REGION Network 92: Step[1902] :
   RUNG wire#powerrail
      { S7_Templates := "SrcType := DInt" } EQ_Contact(in1 := "Unit1.Em2.ControlNodes".semiAutoSplice.sequence.status.currentStep, in2 := #JOB_19_STEP_02)
      Contact( "Unit1.Em2.ControlNodes".semiAutoSplice.sequence.status.seqActive )
      wire#w1
      Coil( "Unit1.Em2.ControlNodes".semiAutoSplice."step".action1[1902] )
   END_RUNG
   RUNG wire#w1
      Coil( "Unit1.Em2.ControlNodes".semiAutoSplice."step".transition1[1902] )
   END_RUNG
   RUNG wire#w1
      Contact( "Unit1.Em2.ControlNodes".semiAutoSplice."step".transition1[1902] )
      { S7_Templates := "time_type := Time" } #statTonTimer[1902].TON(pt := #SeqDelayTime, et =>)
      Move(in := #JOB_19_STEP_03, out1 => "Unit1.Em2.ControlNodes".semiAutoSplice.sequence.status.nextStep)
   END_RUNG
   // the same network as SCL:
   "Unit1.Em2.ControlNodes".semiAutoSplice."step".action1[1902] := ("Unit1.Em2.ControlNodes".semiAutoSplice.sequence.status.currentStep = #JOB_19_STEP_02) AND "Unit1.Em2.ControlNodes".semiAutoSplice.sequence.status.seqActive;
   "Unit1.Em2.ControlNodes".semiAutoSplice."step".transition1[1902] := ("Unit1.Em2.ControlNodes".semiAutoSplice.sequence.status.currentStep = #JOB_19_STEP_02) AND "Unit1.Em2.ControlNodes".semiAutoSplice.sequence.status.seqActive;
   #statTonTimer[1902].TON(IN := ("Unit1.Em2.ControlNodes".semiAutoSplice.sequence.status.currentStep = #JOB_19_STEP_02) AND "Unit1.Em2.ControlNodes".semiAutoSplice.sequence.status.seqActive AND "Unit1.Em2.ControlNodes".semiAutoSplice."step".transition1[1902],
                           PT := #SeqDelayTime);
   IF #statTonTimer[1902].Q THEN
       "Unit1.Em2.ControlNodes".semiAutoSplice.sequence.status.nextStep := #JOB_19_STEP_03;
   END_IF;
END_REGION

REGION Network 93: Step[1903] :
   RUNG wire#powerrail
      { S7_Templates := "SrcType := DInt" } EQ_Contact(in1 := "Unit1.Em2.ControlNodes".semiAutoSplice.sequence.status.currentStep, in2 := #JOB_19_STEP_03)
      Contact( "Unit1.Em2.ControlNodes".semiAutoSplice.sequence.status.seqActive )
      wire#w1
      Coil( "Unit1.Em2.ControlNodes".semiAutoSplice."step".action1[1903] )
   END_RUNG
   RUNG wire#w1
      Coil( "Unit1.Em2.ControlNodes".semiAutoSplice."step".transition1[1903] )
   END_RUNG
   RUNG wire#w1
      Contact( "Unit1.Em2.ControlNodes".semiAutoSplice."step".transition1[1903] )
      { S7_Templates := "time_type := Time" } #statTonTimer[1903].TON(pt := #SeqDelayTime, et =>)
      Move(in := #JOB_19_STEP_04, out1 => "Unit1.Em2.ControlNodes".semiAutoSplice.sequence.status.nextStep)
   END_RUNG
   // the same network as SCL:
   "Unit1.Em2.ControlNodes".semiAutoSplice."step".action1[1903] := ("Unit1.Em2.ControlNodes".semiAutoSplice.sequence.status.currentStep = #JOB_19_STEP_03) AND "Unit1.Em2.ControlNodes".semiAutoSplice.sequence.status.seqActive;
   "Unit1.Em2.ControlNodes".semiAutoSplice."step".transition1[1903] := ("Unit1.Em2.ControlNodes".semiAutoSplice.sequence.status.currentStep = #JOB_19_STEP_03) AND "Unit1.Em2.ControlNodes".semiAutoSplice.sequence.status.seqActive;
   #statTonTimer[1903].TON(IN := ("Unit1.Em2.ControlNodes".semiAutoSplice.sequence.status.currentStep = #JOB_19_STEP_03) AND "Unit1.Em2.ControlNodes".semiAutoSplice.sequence.status.seqActive AND "Unit1.Em2.ControlNodes".semiAutoSplice."step".transition1[1903],
                           PT := #SeqDelayTime);
   IF #statTonTimer[1903].Q THEN
       "Unit1.Em2.ControlNodes".semiAutoSplice.sequence.status.nextStep := #JOB_19_STEP_04;
   END_IF;
END_REGION

REGION Network 94: Step[1904] :
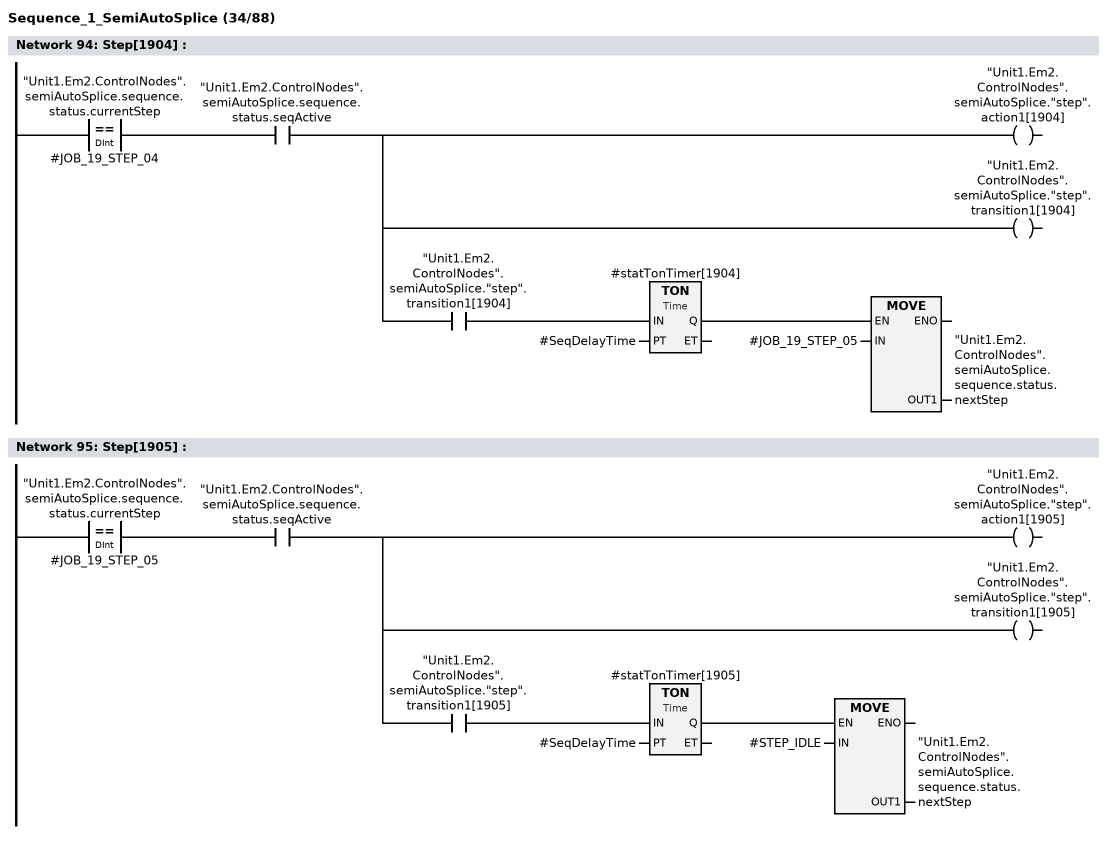
   RUNG wire#powerrail
      { S7_Templates := "SrcType := DInt" } EQ_Contact(in1 := "Unit1.Em2.ControlNodes".semiAutoSplice.sequence.status.currentStep, in2 := #JOB_19_STEP_04)
      Contact( "Unit1.Em2.ControlNodes".semiAutoSplice.sequence.status.seqActive )
      wire#w1
      Coil( "Unit1.Em2.ControlNodes".semiAutoSplice."step".action1[1904] )
   END_RUNG
   RUNG wire#w1
      Coil( "Unit1.Em2.ControlNodes".semiAutoSplice."step".transition1[1904] )
   END_RUNG
   RUNG wire#w1
      Contact( "Unit1.Em2.ControlNodes".semiAutoSplice."step".transition1[1904] )
      { S7_Templates := "time_type := Time" } #statTonTimer[1904].TON(pt := #SeqDelayTime, et =>)
      Move(in := #JOB_19_STEP_05, out1 => "Unit1.Em2.ControlNodes".semiAutoSplice.sequence.status.nextStep)
   END_RUNG
   // the same network as SCL:
   "Unit1.Em2.ControlNodes".semiAutoSplice."step".action1[1904] := ("Unit1.Em2.ControlNodes".semiAutoSplice.sequence.status.currentStep = #JOB_19_STEP_04) AND "Unit1.Em2.ControlNodes".semiAutoSplice.sequence.status.seqActive;
   "Unit1.Em2.ControlNodes".semiAutoSplice."step".transition1[1904] := ("Unit1.Em2.ControlNodes".semiAutoSplice.sequence.status.currentStep = #JOB_19_STEP_04) AND "Unit1.Em2.ControlNodes".semiAutoSplice.sequence.status.seqActive;
   #statTonTimer[1904].TON(IN := ("Unit1.Em2.ControlNodes".semiAutoSplice.sequence.status.currentStep = #JOB_19_STEP_04) AND "Unit1.Em2.ControlNodes".semiAutoSplice.sequence.status.seqActive AND "Unit1.Em2.ControlNodes".semiAutoSplice."step".transition1[1904],
                           PT := #SeqDelayTime);
   IF #statTonTimer[1904].Q THEN
       "Unit1.Em2.ControlNodes".semiAutoSplice.sequence.status.nextStep := #JOB_19_STEP_05;
   END_IF;
END_REGION

REGION Network 95: Step[1905] :
   RUNG wire#powerrail
      { S7_Templates := "SrcType := DInt" } EQ_Contact(in1 := "Unit1.Em2.ControlNodes".semiAutoSplice.sequence.status.currentStep, in2 := #JOB_19_STEP_05)
      Contact( "Unit1.Em2.ControlNodes".semiAutoSplice.sequence.status.seqActive )
      wire#w1
      Coil( "Unit1.Em2.ControlNodes".semiAutoSplice."step".action1[1905] )
   END_RUNG
   RUNG wire#w1
      Coil( "Unit1.Em2.ControlNodes".semiAutoSplice."step".transition1[1905] )
   END_RUNG
   RUNG wire#w1
      Contact( "Unit1.Em2.ControlNodes".semiAutoSplice."step".transition1[1905] )
      { S7_Templates := "time_type := Time" } #statTonTimer[1905].TON(pt := #SeqDelayTime, et =>)
      Move(in := #STEP_IDLE, out1 => "Unit1.Em2.ControlNodes".semiAutoSplice.sequence.status.nextStep)
   END_RUNG
   // the same network as SCL:
   "Unit1.Em2.ControlNodes".semiAutoSplice."step".action1[1905] := ("Unit1.Em2.ControlNodes".semiAutoSplice.sequence.status.currentStep = #JOB_19_STEP_05) AND "Unit1.Em2.ControlNodes".semiAutoSplice.sequence.status.seqActive;
   "Unit1.Em2.ControlNodes".semiAutoSplice."step".transition1[1905] := ("Unit1.Em2.ControlNodes".semiAutoSplice.sequence.status.currentStep = #JOB_19_STEP_05) AND "Unit1.Em2.ControlNodes".semiAutoSplice.sequence.status.seqActive;
   #statTonTimer[1905].TON(IN := ("Unit1.Em2.ControlNodes".semiAutoSplice.sequence.status.currentStep = #JOB_19_STEP_05) AND "Unit1.Em2.ControlNodes".semiAutoSplice.sequence.status.seqActive AND "Unit1.Em2.ControlNodes".semiAutoSplice."step".transition1[1905],
                           PT := #SeqDelayTime);
   IF #statTonTimer[1905].Q THEN
       "Unit1.Em2.ControlNodes".semiAutoSplice.sequence.status.nextStep := #STEP_IDLE;
   END_IF;
END_REGION

REGION Network 96: Step[2001] : Pad Btm Link Btm Left/right Vacc Off (Top Left/Right Vacc On)
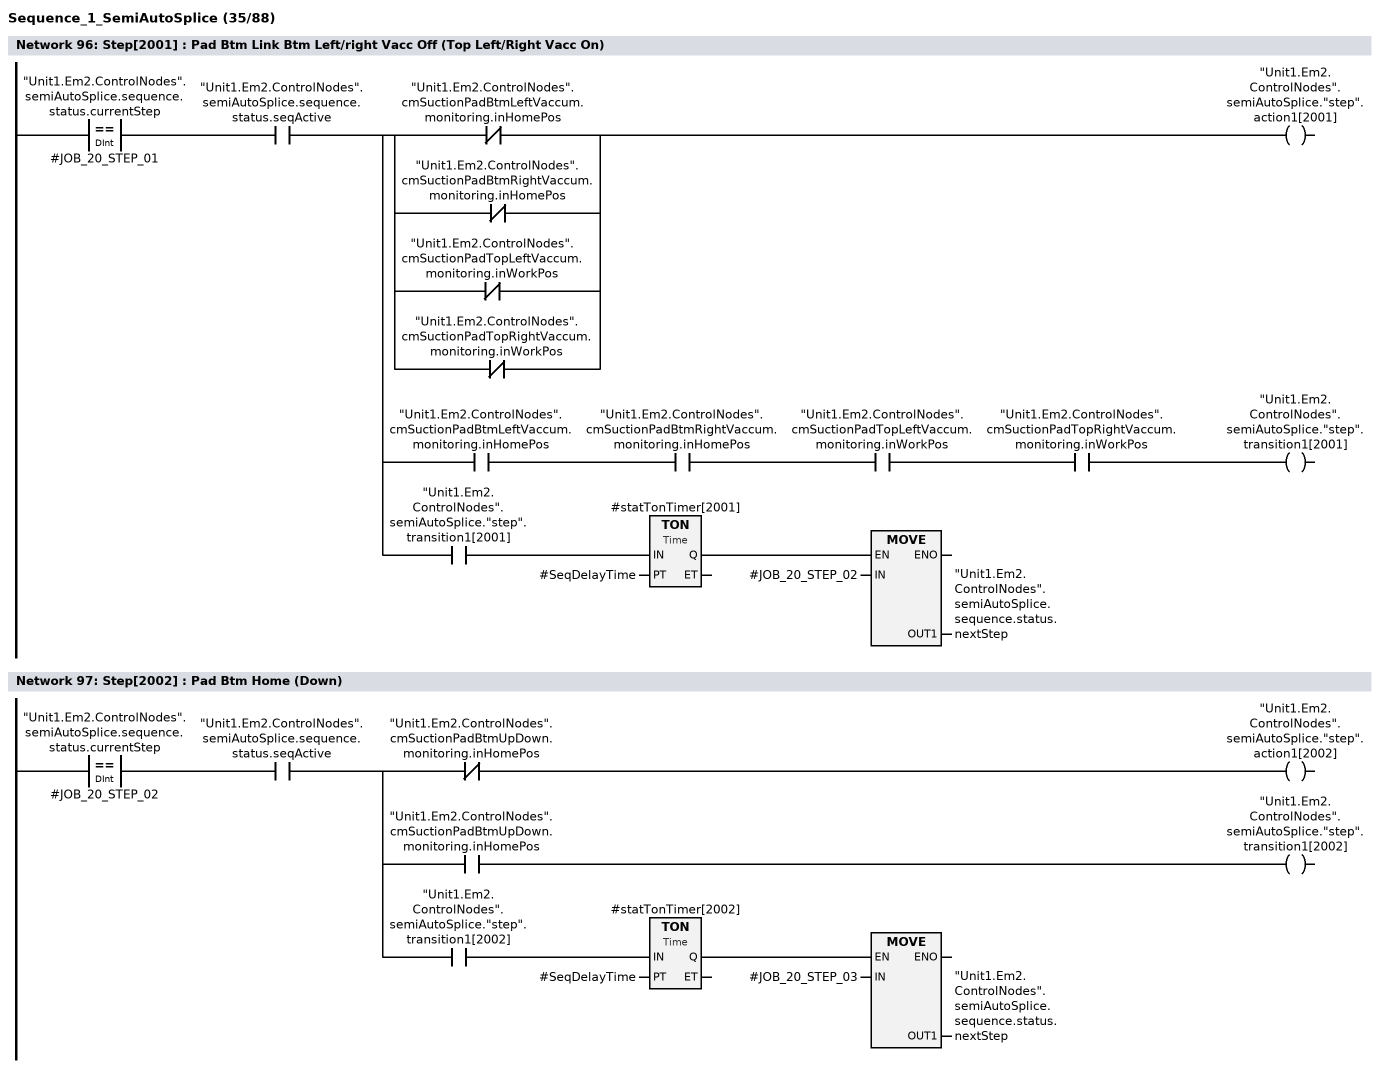
   RUNG wire#powerrail
      { S7_Templates := "SrcType := DInt" } EQ_Contact(in1 := "Unit1.Em2.ControlNodes".semiAutoSplice.sequence.status.currentStep, in2 := #JOB_20_STEP_01)
      Contact( "Unit1.Em2.ControlNodes".semiAutoSplice.sequence.status.seqActive )
      wire#w1
      I_Contact( "Unit1.Em2.ControlNodes".cmSuctionPadBtmLeftVaccum.monitoring.inHomePos )
      wire#w2
      Coil( "Unit1.Em2.ControlNodes".semiAutoSplice."step".action1[2001] )
   END_RUNG
   RUNG wire#w1
      I_Contact( "Unit1.Em2.ControlNodes".cmSuctionPadBtmRightVaccum.monitoring.inHomePos )
   END_RUNG wire#w2
   RUNG wire#w1
      I_Contact( "Unit1.Em2.ControlNodes".cmSuctionPadTopLeftVaccum.monitoring.inWorkPos )
   END_RUNG wire#w2
   RUNG wire#w1
      I_Contact( "Unit1.Em2.ControlNodes".cmSuctionPadTopRightVaccum.monitoring.inWorkPos )
   END_RUNG wire#w2
   RUNG wire#w1
      Contact( "Unit1.Em2.ControlNodes".cmSuctionPadBtmLeftVaccum.monitoring.inHomePos )
      Contact( "Unit1.Em2.ControlNodes".cmSuctionPadBtmRightVaccum.monitoring.inHomePos )
      Contact( "Unit1.Em2.ControlNodes".cmSuctionPadTopLeftVaccum.monitoring.inWorkPos )
      Contact( "Unit1.Em2.ControlNodes".cmSuctionPadTopRightVaccum.monitoring.inWorkPos )
      Coil( "Unit1.Em2.ControlNodes".semiAutoSplice."step".transition1[2001] )
   END_RUNG
   RUNG wire#w1
      Contact( "Unit1.Em2.ControlNodes".semiAutoSplice."step".transition1[2001] )
      { S7_Templates := "time_type := Time" } #statTonTimer[2001].TON(pt := #SeqDelayTime, et =>)
      Move(in := #JOB_20_STEP_02, out1 => "Unit1.Em2.ControlNodes".semiAutoSplice.sequence.status.nextStep)
   END_RUNG
   // the same network as SCL:
   #_w1 := ("Unit1.Em2.ControlNodes".semiAutoSplice.sequence.status.currentStep = #JOB_20_STEP_01) AND "Unit1.Em2.ControlNodes".semiAutoSplice.sequence.status.seqActive;
   "Unit1.Em2.ControlNodes".semiAutoSplice."step".action1[2001] := #_w1 AND (NOT "Unit1.Em2.ControlNodes".cmSuctionPadBtmLeftVaccum.monitoring.inHomePos OR NOT "Unit1.Em2.ControlNodes".cmSuctionPadBtmRightVaccum.monitoring.inHomePos OR NOT "Unit1.Em2.ControlNodes".cmSuctionPadTopLeftVaccum.monitoring.inWorkPos OR NOT "Unit1.Em2.ControlNodes".cmSuctionPadTopRightVaccum.monitoring.inWorkPos);
   "Unit1.Em2.ControlNodes".semiAutoSplice."step".transition1[2001] := #_w1 AND "Unit1.Em2.ControlNodes".cmSuctionPadBtmLeftVaccum.monitoring.inHomePos AND "Unit1.Em2.ControlNodes".cmSuctionPadBtmRightVaccum.monitoring.inHomePos AND "Unit1.Em2.ControlNodes".cmSuctionPadTopLeftVaccum.monitoring.inWorkPos AND "Unit1.Em2.ControlNodes".cmSuctionPadTopRightVaccum.monitoring.inWorkPos;
   #statTonTimer[2001].TON(IN := #_w1 AND "Unit1.Em2.ControlNodes".semiAutoSplice."step".transition1[2001],
                           PT := #SeqDelayTime);
   IF #statTonTimer[2001].Q THEN
       "Unit1.Em2.ControlNodes".semiAutoSplice.sequence.status.nextStep := #JOB_20_STEP_02;
   END_IF;
END_REGION

REGION Network 97: Step[2002] : Pad Btm Home (Down)
   RUNG wire#powerrail
      { S7_Templates := "SrcType := DInt" } EQ_Contact(in1 := "Unit1.Em2.ControlNodes".semiAutoSplice.sequence.status.currentStep, in2 := #JOB_20_STEP_02)
      Contact( "Unit1.Em2.ControlNodes".semiAutoSplice.sequence.status.seqActive )
      wire#w1
      I_Contact( "Unit1.Em2.ControlNodes".cmSuctionPadBtmUpDown.monitoring.inHomePos )
      Coil( "Unit1.Em2.ControlNodes".semiAutoSplice."step".action1[2002] )
   END_RUNG
   RUNG wire#w1
      Contact( "Unit1.Em2.ControlNodes".cmSuctionPadBtmUpDown.monitoring.inHomePos )
      Coil( "Unit1.Em2.ControlNodes".semiAutoSplice."step".transition1[2002] )
   END_RUNG
   RUNG wire#w1
      Contact( "Unit1.Em2.ControlNodes".semiAutoSplice."step".transition1[2002] )
      { S7_Templates := "time_type := Time" } #statTonTimer[2002].TON(pt := #SeqDelayTime, et =>)
      Move(in := #JOB_20_STEP_03, out1 => "Unit1.Em2.ControlNodes".semiAutoSplice.sequence.status.nextStep)
   END_RUNG
   // the same network as SCL:
   #_w1 := ("Unit1.Em2.ControlNodes".semiAutoSplice.sequence.status.currentStep = #JOB_20_STEP_02) AND "Unit1.Em2.ControlNodes".semiAutoSplice.sequence.status.seqActive;
   "Unit1.Em2.ControlNodes".semiAutoSplice."step".action1[2002] := #_w1 AND NOT "Unit1.Em2.ControlNodes".cmSuctionPadBtmUpDown.monitoring.inHomePos;
   "Unit1.Em2.ControlNodes".semiAutoSplice."step".transition1[2002] := #_w1 AND "Unit1.Em2.ControlNodes".cmSuctionPadBtmUpDown.monitoring.inHomePos;
   #statTonTimer[2002].TON(IN := #_w1 AND "Unit1.Em2.ControlNodes".semiAutoSplice."step".transition1[2002],
                           PT := #SeqDelayTime);
   IF #statTonTimer[2002].Q THEN
       "Unit1.Em2.ControlNodes".semiAutoSplice.sequence.status.nextStep := #JOB_20_STEP_03;
   END_IF;
END_REGION

REGION Network 98: Step[2003] :
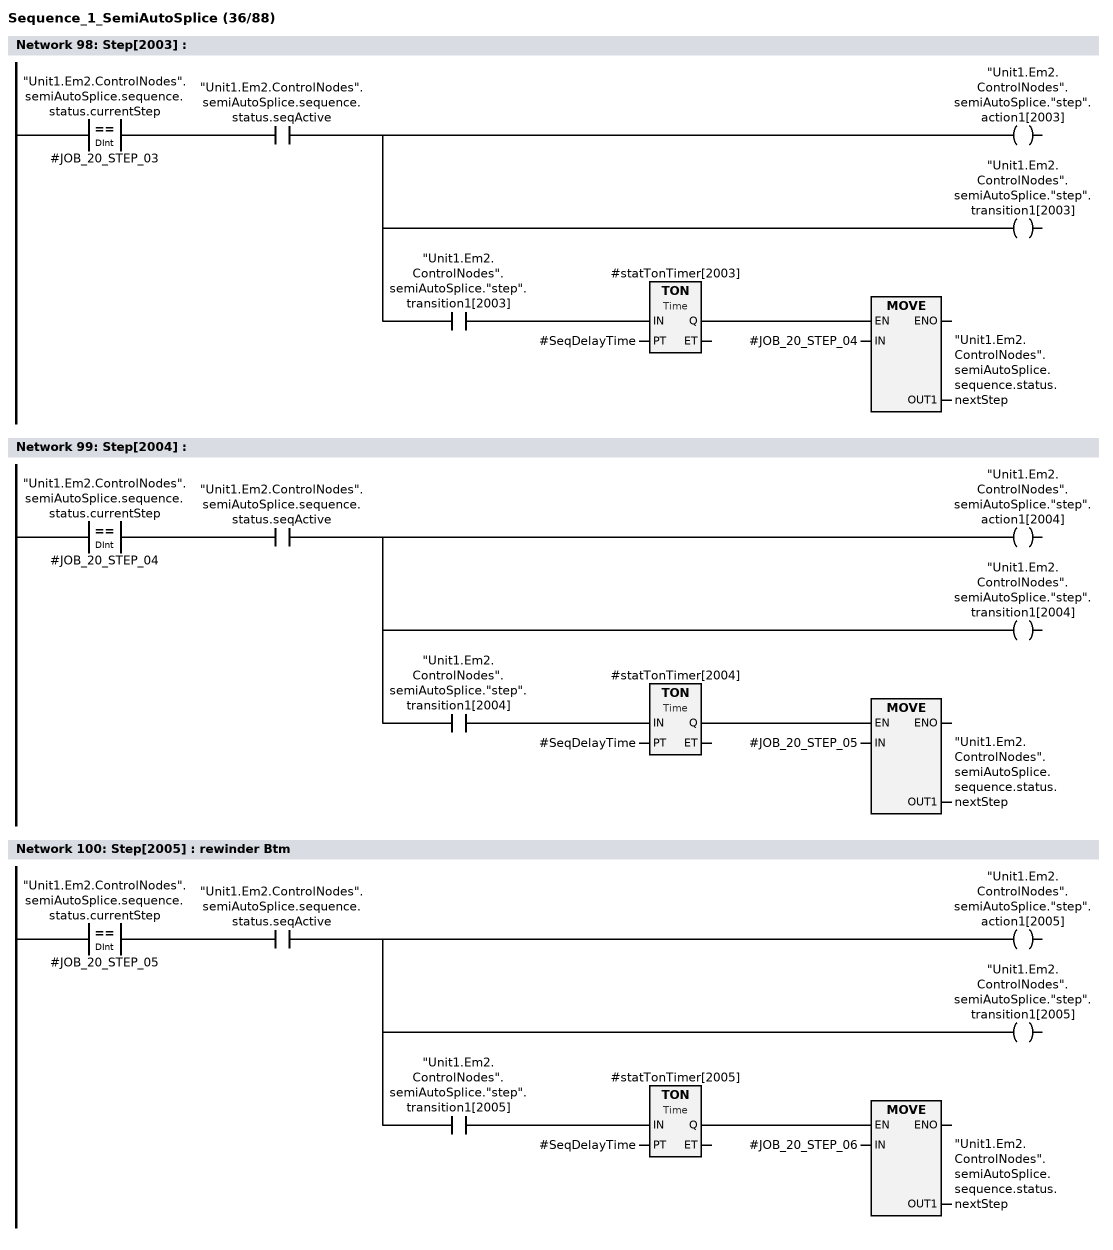
   RUNG wire#powerrail
      { S7_Templates := "SrcType := DInt" } EQ_Contact(in1 := "Unit1.Em2.ControlNodes".semiAutoSplice.sequence.status.currentStep, in2 := #JOB_20_STEP_03)
      Contact( "Unit1.Em2.ControlNodes".semiAutoSplice.sequence.status.seqActive )
      wire#w1
      Coil( "Unit1.Em2.ControlNodes".semiAutoSplice."step".action1[2003] )
   END_RUNG
   RUNG wire#w1
      Coil( "Unit1.Em2.ControlNodes".semiAutoSplice."step".transition1[2003] )
   END_RUNG
   RUNG wire#w1
      Contact( "Unit1.Em2.ControlNodes".semiAutoSplice."step".transition1[2003] )
      { S7_Templates := "time_type := Time" } #statTonTimer[2003].TON(pt := #SeqDelayTime, et =>)
      Move(in := #JOB_20_STEP_04, out1 => "Unit1.Em2.ControlNodes".semiAutoSplice.sequence.status.nextStep)
   END_RUNG
   // the same network as SCL:
   "Unit1.Em2.ControlNodes".semiAutoSplice."step".action1[2003] := ("Unit1.Em2.ControlNodes".semiAutoSplice.sequence.status.currentStep = #JOB_20_STEP_03) AND "Unit1.Em2.ControlNodes".semiAutoSplice.sequence.status.seqActive;
   "Unit1.Em2.ControlNodes".semiAutoSplice."step".transition1[2003] := ("Unit1.Em2.ControlNodes".semiAutoSplice.sequence.status.currentStep = #JOB_20_STEP_03) AND "Unit1.Em2.ControlNodes".semiAutoSplice.sequence.status.seqActive;
   #statTonTimer[2003].TON(IN := ("Unit1.Em2.ControlNodes".semiAutoSplice.sequence.status.currentStep = #JOB_20_STEP_03) AND "Unit1.Em2.ControlNodes".semiAutoSplice.sequence.status.seqActive AND "Unit1.Em2.ControlNodes".semiAutoSplice."step".transition1[2003],
                           PT := #SeqDelayTime);
   IF #statTonTimer[2003].Q THEN
       "Unit1.Em2.ControlNodes".semiAutoSplice.sequence.status.nextStep := #JOB_20_STEP_04;
   END_IF;
END_REGION

REGION Network 99: Step[2004] :
   RUNG wire#powerrail
      { S7_Templates := "SrcType := DInt" } EQ_Contact(in1 := "Unit1.Em2.ControlNodes".semiAutoSplice.sequence.status.currentStep, in2 := #JOB_20_STEP_04)
      Contact( "Unit1.Em2.ControlNodes".semiAutoSplice.sequence.status.seqActive )
      wire#w1
      Coil( "Unit1.Em2.ControlNodes".semiAutoSplice."step".action1[2004] )
   END_RUNG
   RUNG wire#w1
      Coil( "Unit1.Em2.ControlNodes".semiAutoSplice."step".transition1[2004] )
   END_RUNG
   RUNG wire#w1
      Contact( "Unit1.Em2.ControlNodes".semiAutoSplice."step".transition1[2004] )
      { S7_Templates := "time_type := Time" } #statTonTimer[2004].TON(pt := #SeqDelayTime, et =>)
      Move(in := #JOB_20_STEP_05, out1 => "Unit1.Em2.ControlNodes".semiAutoSplice.sequence.status.nextStep)
   END_RUNG
   // the same network as SCL:
   "Unit1.Em2.ControlNodes".semiAutoSplice."step".action1[2004] := ("Unit1.Em2.ControlNodes".semiAutoSplice.sequence.status.currentStep = #JOB_20_STEP_04) AND "Unit1.Em2.ControlNodes".semiAutoSplice.sequence.status.seqActive;
   "Unit1.Em2.ControlNodes".semiAutoSplice."step".transition1[2004] := ("Unit1.Em2.ControlNodes".semiAutoSplice.sequence.status.currentStep = #JOB_20_STEP_04) AND "Unit1.Em2.ControlNodes".semiAutoSplice.sequence.status.seqActive;
   #statTonTimer[2004].TON(IN := ("Unit1.Em2.ControlNodes".semiAutoSplice.sequence.status.currentStep = #JOB_20_STEP_04) AND "Unit1.Em2.ControlNodes".semiAutoSplice.sequence.status.seqActive AND "Unit1.Em2.ControlNodes".semiAutoSplice."step".transition1[2004],
                           PT := #SeqDelayTime);
   IF #statTonTimer[2004].Q THEN
       "Unit1.Em2.ControlNodes".semiAutoSplice.sequence.status.nextStep := #JOB_20_STEP_05;
   END_IF;
END_REGION

REGION Network 100: Step[2005] : rewinder Btm
   RUNG wire#powerrail
      { S7_Templates := "SrcType := DInt" } EQ_Contact(in1 := "Unit1.Em2.ControlNodes".semiAutoSplice.sequence.status.currentStep, in2 := #JOB_20_STEP_05)
      Contact( "Unit1.Em2.ControlNodes".semiAutoSplice.sequence.status.seqActive )
      wire#w1
      Coil( "Unit1.Em2.ControlNodes".semiAutoSplice."step".action1[2005] )
   END_RUNG
   RUNG wire#w1
      Coil( "Unit1.Em2.ControlNodes".semiAutoSplice."step".transition1[2005] )
   END_RUNG
   RUNG wire#w1
      Contact( "Unit1.Em2.ControlNodes".semiAutoSplice."step".transition1[2005] )
      { S7_Templates := "time_type := Time" } #statTonTimer[2005].TON(pt := #SeqDelayTime, et =>)
      Move(in := #JOB_20_STEP_06, out1 => "Unit1.Em2.ControlNodes".semiAutoSplice.sequence.status.nextStep)
   END_RUNG
   // the same network as SCL:
   "Unit1.Em2.ControlNodes".semiAutoSplice."step".action1[2005] := ("Unit1.Em2.ControlNodes".semiAutoSplice.sequence.status.currentStep = #JOB_20_STEP_05) AND "Unit1.Em2.ControlNodes".semiAutoSplice.sequence.status.seqActive;
   "Unit1.Em2.ControlNodes".semiAutoSplice."step".transition1[2005] := ("Unit1.Em2.ControlNodes".semiAutoSplice.sequence.status.currentStep = #JOB_20_STEP_05) AND "Unit1.Em2.ControlNodes".semiAutoSplice.sequence.status.seqActive;
   #statTonTimer[2005].TON(IN := ("Unit1.Em2.ControlNodes".semiAutoSplice.sequence.status.currentStep = #JOB_20_STEP_05) AND "Unit1.Em2.ControlNodes".semiAutoSplice.sequence.status.seqActive AND "Unit1.Em2.ControlNodes".semiAutoSplice."step".transition1[2005],
                           PT := #SeqDelayTime);
   IF #statTonTimer[2005].Q THEN
       "Unit1.Em2.ControlNodes".semiAutoSplice.sequence.status.nextStep := #JOB_20_STEP_06;
   END_IF;
END_REGION

REGION Network 101: Step[2006] : Complete
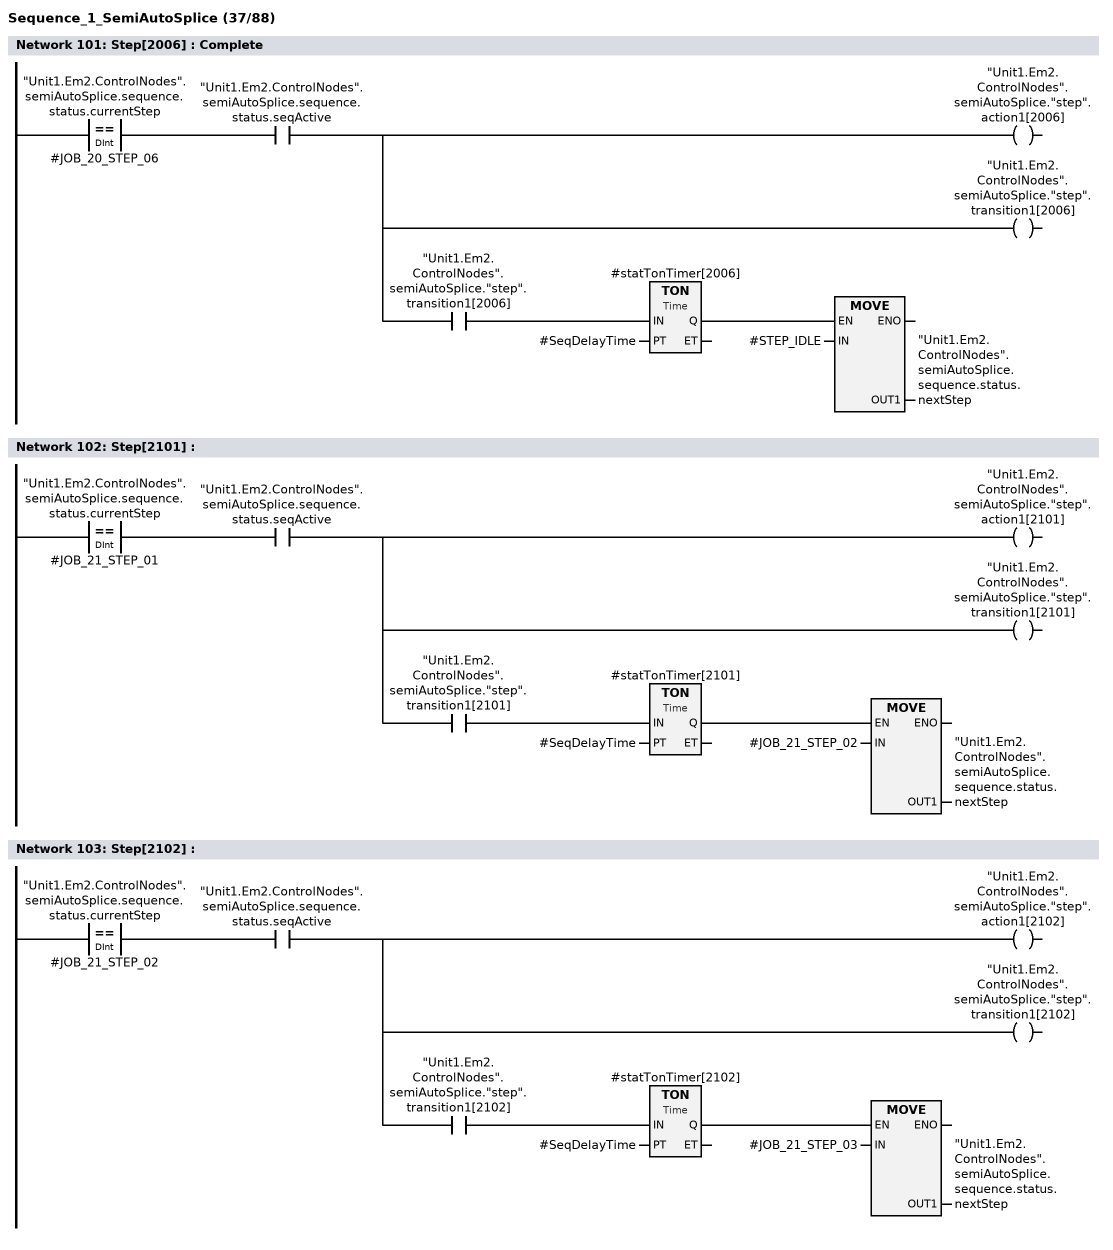
   RUNG wire#powerrail
      { S7_Templates := "SrcType := DInt" } EQ_Contact(in1 := "Unit1.Em2.ControlNodes".semiAutoSplice.sequence.status.currentStep, in2 := #JOB_20_STEP_06)
      Contact( "Unit1.Em2.ControlNodes".semiAutoSplice.sequence.status.seqActive )
      wire#w1
      Coil( "Unit1.Em2.ControlNodes".semiAutoSplice."step".action1[2006] )
   END_RUNG
   RUNG wire#w1
      Coil( "Unit1.Em2.ControlNodes".semiAutoSplice."step".transition1[2006] )
   END_RUNG
   RUNG wire#w1
      Contact( "Unit1.Em2.ControlNodes".semiAutoSplice."step".transition1[2006] )
      { S7_Templates := "time_type := Time" } #statTonTimer[2006].TON(pt := #SeqDelayTime, et =>)
      Move(in := #STEP_IDLE, out1 => "Unit1.Em2.ControlNodes".semiAutoSplice.sequence.status.nextStep)
   END_RUNG
   // the same network as SCL:
   "Unit1.Em2.ControlNodes".semiAutoSplice."step".action1[2006] := ("Unit1.Em2.ControlNodes".semiAutoSplice.sequence.status.currentStep = #JOB_20_STEP_06) AND "Unit1.Em2.ControlNodes".semiAutoSplice.sequence.status.seqActive;
   "Unit1.Em2.ControlNodes".semiAutoSplice."step".transition1[2006] := ("Unit1.Em2.ControlNodes".semiAutoSplice.sequence.status.currentStep = #JOB_20_STEP_06) AND "Unit1.Em2.ControlNodes".semiAutoSplice.sequence.status.seqActive;
   #statTonTimer[2006].TON(IN := ("Unit1.Em2.ControlNodes".semiAutoSplice.sequence.status.currentStep = #JOB_20_STEP_06) AND "Unit1.Em2.ControlNodes".semiAutoSplice.sequence.status.seqActive AND "Unit1.Em2.ControlNodes".semiAutoSplice."step".transition1[2006],
                           PT := #SeqDelayTime);
   IF #statTonTimer[2006].Q THEN
       "Unit1.Em2.ControlNodes".semiAutoSplice.sequence.status.nextStep := #STEP_IDLE;
   END_IF;
END_REGION

REGION Network 102: Step[2101] :
   RUNG wire#powerrail
      { S7_Templates := "SrcType := DInt" } EQ_Contact(in1 := "Unit1.Em2.ControlNodes".semiAutoSplice.sequence.status.currentStep, in2 := #JOB_21_STEP_01)
      Contact( "Unit1.Em2.ControlNodes".semiAutoSplice.sequence.status.seqActive )
      wire#w1
      Coil( "Unit1.Em2.ControlNodes".semiAutoSplice."step".action1[2101] )
   END_RUNG
   RUNG wire#w1
      Coil( "Unit1.Em2.ControlNodes".semiAutoSplice."step".transition1[2101] )
   END_RUNG
   RUNG wire#w1
      Contact( "Unit1.Em2.ControlNodes".semiAutoSplice."step".transition1[2101] )
      { S7_Templates := "time_type := Time" } #statTonTimer[2101].TON(pt := #SeqDelayTime, et =>)
      Move(in := #JOB_21_STEP_02, out1 => "Unit1.Em2.ControlNodes".semiAutoSplice.sequence.status.nextStep)
   END_RUNG
   // the same network as SCL:
   "Unit1.Em2.ControlNodes".semiAutoSplice."step".action1[2101] := ("Unit1.Em2.ControlNodes".semiAutoSplice.sequence.status.currentStep = #JOB_21_STEP_01) AND "Unit1.Em2.ControlNodes".semiAutoSplice.sequence.status.seqActive;
   "Unit1.Em2.ControlNodes".semiAutoSplice."step".transition1[2101] := ("Unit1.Em2.ControlNodes".semiAutoSplice.sequence.status.currentStep = #JOB_21_STEP_01) AND "Unit1.Em2.ControlNodes".semiAutoSplice.sequence.status.seqActive;
   #statTonTimer[2101].TON(IN := ("Unit1.Em2.ControlNodes".semiAutoSplice.sequence.status.currentStep = #JOB_21_STEP_01) AND "Unit1.Em2.ControlNodes".semiAutoSplice.sequence.status.seqActive AND "Unit1.Em2.ControlNodes".semiAutoSplice."step".transition1[2101],
                           PT := #SeqDelayTime);
   IF #statTonTimer[2101].Q THEN
       "Unit1.Em2.ControlNodes".semiAutoSplice.sequence.status.nextStep := #JOB_21_STEP_02;
   END_IF;
END_REGION

REGION Network 103: Step[2102] :
   RUNG wire#powerrail
      { S7_Templates := "SrcType := DInt" } EQ_Contact(in1 := "Unit1.Em2.ControlNodes".semiAutoSplice.sequence.status.currentStep, in2 := #JOB_21_STEP_02)
      Contact( "Unit1.Em2.ControlNodes".semiAutoSplice.sequence.status.seqActive )
      wire#w1
      Coil( "Unit1.Em2.ControlNodes".semiAutoSplice."step".action1[2102] )
   END_RUNG
   RUNG wire#w1
      Coil( "Unit1.Em2.ControlNodes".semiAutoSplice."step".transition1[2102] )
   END_RUNG
   RUNG wire#w1
      Contact( "Unit1.Em2.ControlNodes".semiAutoSplice."step".transition1[2102] )
      { S7_Templates := "time_type := Time" } #statTonTimer[2102].TON(pt := #SeqDelayTime, et =>)
      Move(in := #JOB_21_STEP_03, out1 => "Unit1.Em2.ControlNodes".semiAutoSplice.sequence.status.nextStep)
   END_RUNG
   // the same network as SCL:
   "Unit1.Em2.ControlNodes".semiAutoSplice."step".action1[2102] := ("Unit1.Em2.ControlNodes".semiAutoSplice.sequence.status.currentStep = #JOB_21_STEP_02) AND "Unit1.Em2.ControlNodes".semiAutoSplice.sequence.status.seqActive;
   "Unit1.Em2.ControlNodes".semiAutoSplice."step".transition1[2102] := ("Unit1.Em2.ControlNodes".semiAutoSplice.sequence.status.currentStep = #JOB_21_STEP_02) AND "Unit1.Em2.ControlNodes".semiAutoSplice.sequence.status.seqActive;
   #statTonTimer[2102].TON(IN := ("Unit1.Em2.ControlNodes".semiAutoSplice.sequence.status.currentStep = #JOB_21_STEP_02) AND "Unit1.Em2.ControlNodes".semiAutoSplice.sequence.status.seqActive AND "Unit1.Em2.ControlNodes".semiAutoSplice."step".transition1[2102],
                           PT := #SeqDelayTime);
   IF #statTonTimer[2102].Q THEN
       "Unit1.Em2.ControlNodes".semiAutoSplice.sequence.status.nextStep := #JOB_21_STEP_03;
   END_IF;
END_REGION

REGION Network 104: Step[2103] :
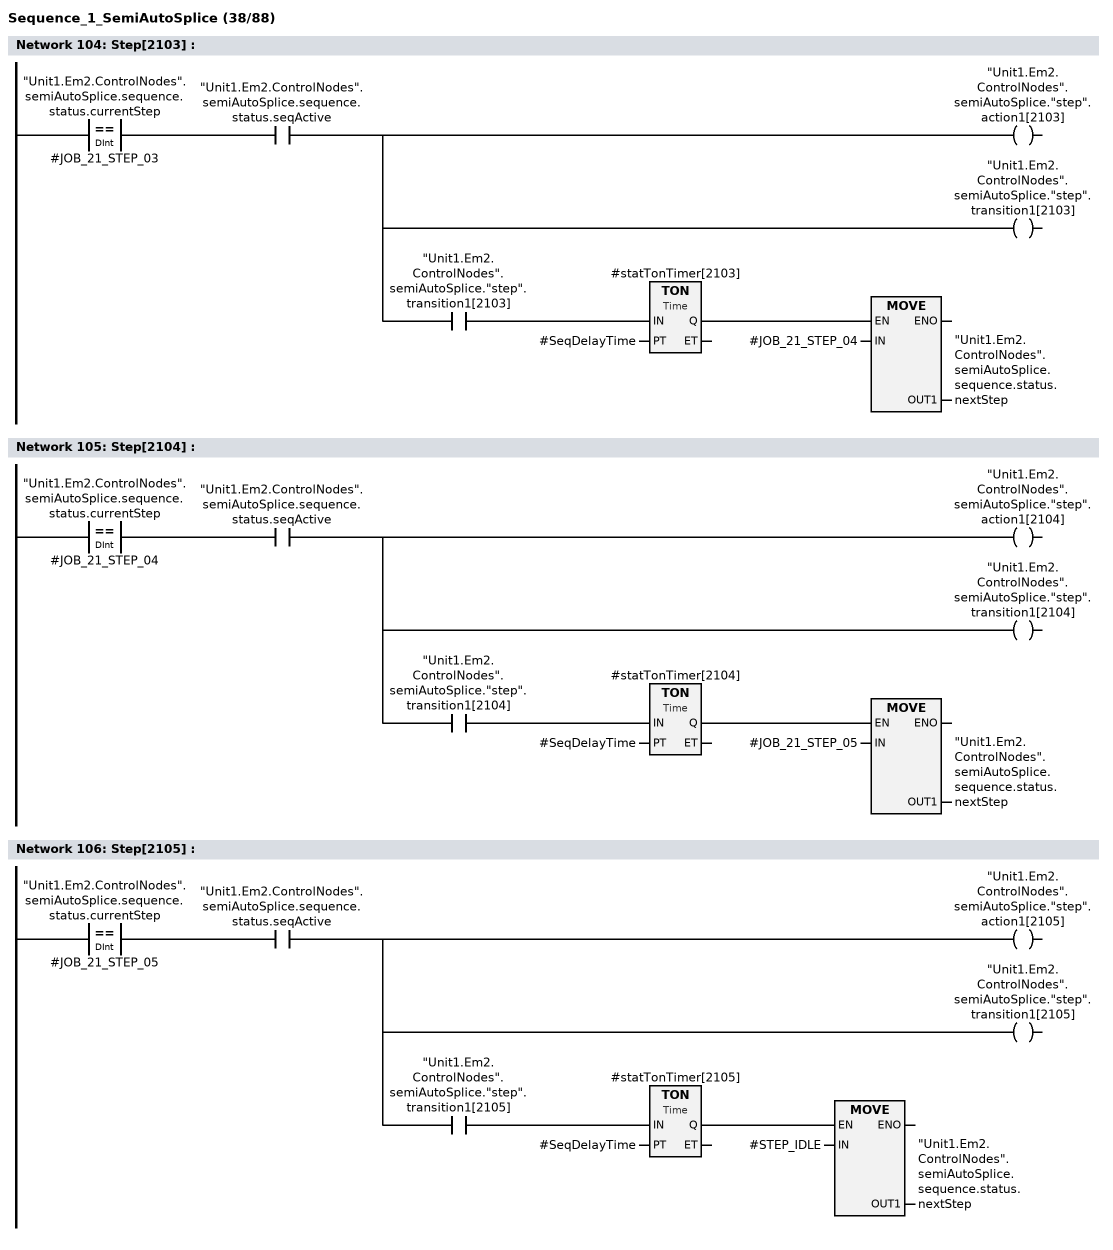
   RUNG wire#powerrail
      { S7_Templates := "SrcType := DInt" } EQ_Contact(in1 := "Unit1.Em2.ControlNodes".semiAutoSplice.sequence.status.currentStep, in2 := #JOB_21_STEP_03)
      Contact( "Unit1.Em2.ControlNodes".semiAutoSplice.sequence.status.seqActive )
      wire#w1
      Coil( "Unit1.Em2.ControlNodes".semiAutoSplice."step".action1[2103] )
   END_RUNG
   RUNG wire#w1
      Coil( "Unit1.Em2.ControlNodes".semiAutoSplice."step".transition1[2103] )
   END_RUNG
   RUNG wire#w1
      Contact( "Unit1.Em2.ControlNodes".semiAutoSplice."step".transition1[2103] )
      { S7_Templates := "time_type := Time" } #statTonTimer[2103].TON(pt := #SeqDelayTime, et =>)
      Move(in := #JOB_21_STEP_04, out1 => "Unit1.Em2.ControlNodes".semiAutoSplice.sequence.status.nextStep)
   END_RUNG
   // the same network as SCL:
   "Unit1.Em2.ControlNodes".semiAutoSplice."step".action1[2103] := ("Unit1.Em2.ControlNodes".semiAutoSplice.sequence.status.currentStep = #JOB_21_STEP_03) AND "Unit1.Em2.ControlNodes".semiAutoSplice.sequence.status.seqActive;
   "Unit1.Em2.ControlNodes".semiAutoSplice."step".transition1[2103] := ("Unit1.Em2.ControlNodes".semiAutoSplice.sequence.status.currentStep = #JOB_21_STEP_03) AND "Unit1.Em2.ControlNodes".semiAutoSplice.sequence.status.seqActive;
   #statTonTimer[2103].TON(IN := ("Unit1.Em2.ControlNodes".semiAutoSplice.sequence.status.currentStep = #JOB_21_STEP_03) AND "Unit1.Em2.ControlNodes".semiAutoSplice.sequence.status.seqActive AND "Unit1.Em2.ControlNodes".semiAutoSplice."step".transition1[2103],
                           PT := #SeqDelayTime);
   IF #statTonTimer[2103].Q THEN
       "Unit1.Em2.ControlNodes".semiAutoSplice.sequence.status.nextStep := #JOB_21_STEP_04;
   END_IF;
END_REGION

REGION Network 105: Step[2104] :
   RUNG wire#powerrail
      { S7_Templates := "SrcType := DInt" } EQ_Contact(in1 := "Unit1.Em2.ControlNodes".semiAutoSplice.sequence.status.currentStep, in2 := #JOB_21_STEP_04)
      Contact( "Unit1.Em2.ControlNodes".semiAutoSplice.sequence.status.seqActive )
      wire#w1
      Coil( "Unit1.Em2.ControlNodes".semiAutoSplice."step".action1[2104] )
   END_RUNG
   RUNG wire#w1
      Coil( "Unit1.Em2.ControlNodes".semiAutoSplice."step".transition1[2104] )
   END_RUNG
   RUNG wire#w1
      Contact( "Unit1.Em2.ControlNodes".semiAutoSplice."step".transition1[2104] )
      { S7_Templates := "time_type := Time" } #statTonTimer[2104].TON(pt := #SeqDelayTime, et =>)
      Move(in := #JOB_21_STEP_05, out1 => "Unit1.Em2.ControlNodes".semiAutoSplice.sequence.status.nextStep)
   END_RUNG
   // the same network as SCL:
   "Unit1.Em2.ControlNodes".semiAutoSplice."step".action1[2104] := ("Unit1.Em2.ControlNodes".semiAutoSplice.sequence.status.currentStep = #JOB_21_STEP_04) AND "Unit1.Em2.ControlNodes".semiAutoSplice.sequence.status.seqActive;
   "Unit1.Em2.ControlNodes".semiAutoSplice."step".transition1[2104] := ("Unit1.Em2.ControlNodes".semiAutoSplice.sequence.status.currentStep = #JOB_21_STEP_04) AND "Unit1.Em2.ControlNodes".semiAutoSplice.sequence.status.seqActive;
   #statTonTimer[2104].TON(IN := ("Unit1.Em2.ControlNodes".semiAutoSplice.sequence.status.currentStep = #JOB_21_STEP_04) AND "Unit1.Em2.ControlNodes".semiAutoSplice.sequence.status.seqActive AND "Unit1.Em2.ControlNodes".semiAutoSplice."step".transition1[2104],
                           PT := #SeqDelayTime);
   IF #statTonTimer[2104].Q THEN
       "Unit1.Em2.ControlNodes".semiAutoSplice.sequence.status.nextStep := #JOB_21_STEP_05;
   END_IF;
END_REGION

REGION Network 106: Step[2105] :
   RUNG wire#powerrail
      { S7_Templates := "SrcType := DInt" } EQ_Contact(in1 := "Unit1.Em2.ControlNodes".semiAutoSplice.sequence.status.currentStep, in2 := #JOB_21_STEP_05)
      Contact( "Unit1.Em2.ControlNodes".semiAutoSplice.sequence.status.seqActive )
      wire#w1
      Coil( "Unit1.Em2.ControlNodes".semiAutoSplice."step".action1[2105] )
   END_RUNG
   RUNG wire#w1
      Coil( "Unit1.Em2.ControlNodes".semiAutoSplice."step".transition1[2105] )
   END_RUNG
   RUNG wire#w1
      Contact( "Unit1.Em2.ControlNodes".semiAutoSplice."step".transition1[2105] )
      { S7_Templates := "time_type := Time" } #statTonTimer[2105].TON(pt := #SeqDelayTime, et =>)
      Move(in := #STEP_IDLE, out1 => "Unit1.Em2.ControlNodes".semiAutoSplice.sequence.status.nextStep)
   END_RUNG
   // the same network as SCL:
   "Unit1.Em2.ControlNodes".semiAutoSplice."step".action1[2105] := ("Unit1.Em2.ControlNodes".semiAutoSplice.sequence.status.currentStep = #JOB_21_STEP_05) AND "Unit1.Em2.ControlNodes".semiAutoSplice.sequence.status.seqActive;
   "Unit1.Em2.ControlNodes".semiAutoSplice."step".transition1[2105] := ("Unit1.Em2.ControlNodes".semiAutoSplice.sequence.status.currentStep = #JOB_21_STEP_05) AND "Unit1.Em2.ControlNodes".semiAutoSplice.sequence.status.seqActive;
   #statTonTimer[2105].TON(IN := ("Unit1.Em2.ControlNodes".semiAutoSplice.sequence.status.currentStep = #JOB_21_STEP_05) AND "Unit1.Em2.ControlNodes".semiAutoSplice.sequence.status.seqActive AND "Unit1.Em2.ControlNodes".semiAutoSplice."step".transition1[2105],
                           PT := #SeqDelayTime);
   IF #statTonTimer[2105].Q THEN
       "Unit1.Em2.ControlNodes".semiAutoSplice.sequence.status.nextStep := #STEP_IDLE;
   END_IF;
END_REGION

REGION Network 107: Step[2201] : Pad Btm Work (Up)
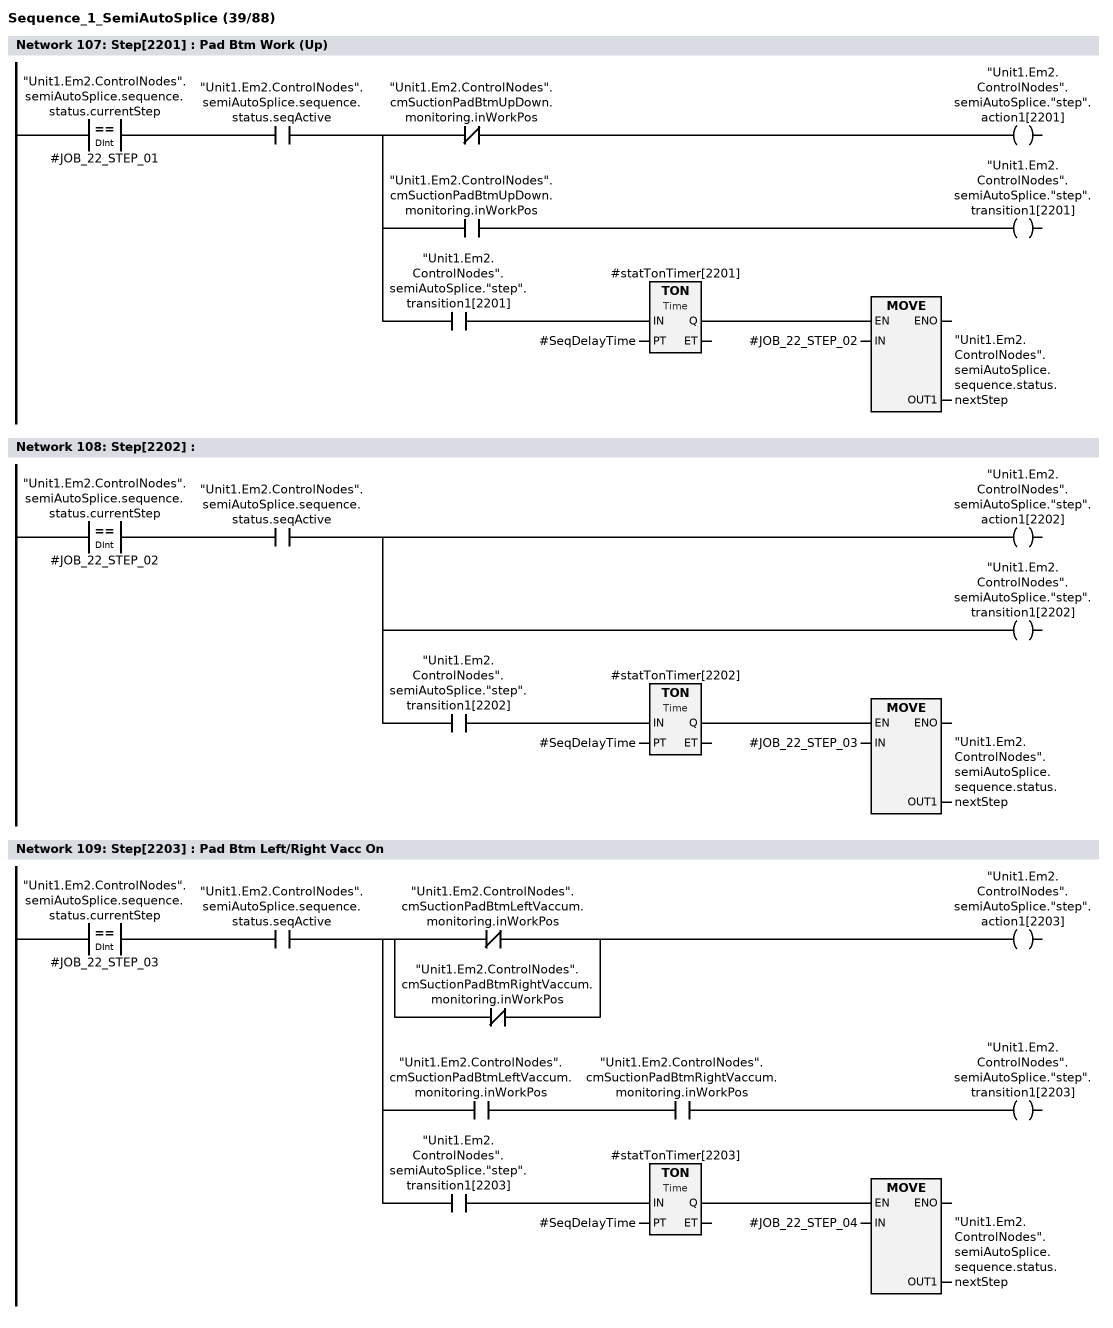
   RUNG wire#powerrail
      { S7_Templates := "SrcType := DInt" } EQ_Contact(in1 := "Unit1.Em2.ControlNodes".semiAutoSplice.sequence.status.currentStep, in2 := #JOB_22_STEP_01)
      Contact( "Unit1.Em2.ControlNodes".semiAutoSplice.sequence.status.seqActive )
      wire#w1
      I_Contact( "Unit1.Em2.ControlNodes".cmSuctionPadBtmUpDown.monitoring.inWorkPos )
      Coil( "Unit1.Em2.ControlNodes".semiAutoSplice."step".action1[2201] )
   END_RUNG
   RUNG wire#w1
      Contact( "Unit1.Em2.ControlNodes".cmSuctionPadBtmUpDown.monitoring.inWorkPos )
      Coil( "Unit1.Em2.ControlNodes".semiAutoSplice."step".transition1[2201] )
   END_RUNG
   RUNG wire#w1
      Contact( "Unit1.Em2.ControlNodes".semiAutoSplice."step".transition1[2201] )
      { S7_Templates := "time_type := Time" } #statTonTimer[2201].TON(pt := #SeqDelayTime, et =>)
      Move(in := #JOB_22_STEP_02, out1 => "Unit1.Em2.ControlNodes".semiAutoSplice.sequence.status.nextStep)
   END_RUNG
   // the same network as SCL:
   #_w1 := ("Unit1.Em2.ControlNodes".semiAutoSplice.sequence.status.currentStep = #JOB_22_STEP_01) AND "Unit1.Em2.ControlNodes".semiAutoSplice.sequence.status.seqActive;
   "Unit1.Em2.ControlNodes".semiAutoSplice."step".action1[2201] := #_w1 AND NOT "Unit1.Em2.ControlNodes".cmSuctionPadBtmUpDown.monitoring.inWorkPos;
   "Unit1.Em2.ControlNodes".semiAutoSplice."step".transition1[2201] := #_w1 AND "Unit1.Em2.ControlNodes".cmSuctionPadBtmUpDown.monitoring.inWorkPos;
   #statTonTimer[2201].TON(IN := #_w1 AND "Unit1.Em2.ControlNodes".semiAutoSplice."step".transition1[2201],
                           PT := #SeqDelayTime);
   IF #statTonTimer[2201].Q THEN
       "Unit1.Em2.ControlNodes".semiAutoSplice.sequence.status.nextStep := #JOB_22_STEP_02;
   END_IF;
END_REGION

REGION Network 108: Step[2202] :
   RUNG wire#powerrail
      { S7_Templates := "SrcType := DInt" } EQ_Contact(in1 := "Unit1.Em2.ControlNodes".semiAutoSplice.sequence.status.currentStep, in2 := #JOB_22_STEP_02)
      Contact( "Unit1.Em2.ControlNodes".semiAutoSplice.sequence.status.seqActive )
      wire#w1
      Coil( "Unit1.Em2.ControlNodes".semiAutoSplice."step".action1[2202] )
   END_RUNG
   RUNG wire#w1
      Coil( "Unit1.Em2.ControlNodes".semiAutoSplice."step".transition1[2202] )
   END_RUNG
   RUNG wire#w1
      Contact( "Unit1.Em2.ControlNodes".semiAutoSplice."step".transition1[2202] )
      { S7_Templates := "time_type := Time" } #statTonTimer[2202].TON(pt := #SeqDelayTime, et =>)
      Move(in := #JOB_22_STEP_03, out1 => "Unit1.Em2.ControlNodes".semiAutoSplice.sequence.status.nextStep)
   END_RUNG
   // the same network as SCL:
   "Unit1.Em2.ControlNodes".semiAutoSplice."step".action1[2202] := ("Unit1.Em2.ControlNodes".semiAutoSplice.sequence.status.currentStep = #JOB_22_STEP_02) AND "Unit1.Em2.ControlNodes".semiAutoSplice.sequence.status.seqActive;
   "Unit1.Em2.ControlNodes".semiAutoSplice."step".transition1[2202] := ("Unit1.Em2.ControlNodes".semiAutoSplice.sequence.status.currentStep = #JOB_22_STEP_02) AND "Unit1.Em2.ControlNodes".semiAutoSplice.sequence.status.seqActive;
   #statTonTimer[2202].TON(IN := ("Unit1.Em2.ControlNodes".semiAutoSplice.sequence.status.currentStep = #JOB_22_STEP_02) AND "Unit1.Em2.ControlNodes".semiAutoSplice.sequence.status.seqActive AND "Unit1.Em2.ControlNodes".semiAutoSplice."step".transition1[2202],
                           PT := #SeqDelayTime);
   IF #statTonTimer[2202].Q THEN
       "Unit1.Em2.ControlNodes".semiAutoSplice.sequence.status.nextStep := #JOB_22_STEP_03;
   END_IF;
END_REGION

REGION Network 109: Step[2203] : Pad Btm Left/Right Vacc On
   RUNG wire#powerrail
      { S7_Templates := "SrcType := DInt" } EQ_Contact(in1 := "Unit1.Em2.ControlNodes".semiAutoSplice.sequence.status.currentStep, in2 := #JOB_22_STEP_03)
      Contact( "Unit1.Em2.ControlNodes".semiAutoSplice.sequence.status.seqActive )
      wire#w1
      I_Contact( "Unit1.Em2.ControlNodes".cmSuctionPadBtmLeftVaccum.monitoring.inWorkPos )
      wire#w2
      Coil( "Unit1.Em2.ControlNodes".semiAutoSplice."step".action1[2203] )
   END_RUNG
   RUNG wire#w1
      I_Contact( "Unit1.Em2.ControlNodes".cmSuctionPadBtmRightVaccum.monitoring.inWorkPos )
   END_RUNG wire#w2
   RUNG wire#w1
      Contact( "Unit1.Em2.ControlNodes".cmSuctionPadBtmLeftVaccum.monitoring.inWorkPos )
      Contact( "Unit1.Em2.ControlNodes".cmSuctionPadBtmRightVaccum.monitoring.inWorkPos )
      Coil( "Unit1.Em2.ControlNodes".semiAutoSplice."step".transition1[2203] )
   END_RUNG
   RUNG wire#w1
      Contact( "Unit1.Em2.ControlNodes".semiAutoSplice."step".transition1[2203] )
      { S7_Templates := "time_type := Time" } #statTonTimer[2203].TON(pt := #SeqDelayTime, et =>)
      Move(in := #JOB_22_STEP_04, out1 => "Unit1.Em2.ControlNodes".semiAutoSplice.sequence.status.nextStep)
   END_RUNG
   // the same network as SCL:
   #_w1 := ("Unit1.Em2.ControlNodes".semiAutoSplice.sequence.status.currentStep = #JOB_22_STEP_03) AND "Unit1.Em2.ControlNodes".semiAutoSplice.sequence.status.seqActive;
   "Unit1.Em2.ControlNodes".semiAutoSplice."step".action1[2203] := #_w1 AND (NOT "Unit1.Em2.ControlNodes".cmSuctionPadBtmLeftVaccum.monitoring.inWorkPos OR NOT "Unit1.Em2.ControlNodes".cmSuctionPadBtmRightVaccum.monitoring.inWorkPos);
   "Unit1.Em2.ControlNodes".semiAutoSplice."step".transition1[2203] := #_w1 AND "Unit1.Em2.ControlNodes".cmSuctionPadBtmLeftVaccum.monitoring.inWorkPos AND "Unit1.Em2.ControlNodes".cmSuctionPadBtmRightVaccum.monitoring.inWorkPos;
   #statTonTimer[2203].TON(IN := #_w1 AND "Unit1.Em2.ControlNodes".semiAutoSplice."step".transition1[2203],
                           PT := #SeqDelayTime);
   IF #statTonTimer[2203].Q THEN
       "Unit1.Em2.ControlNodes".semiAutoSplice.sequence.status.nextStep := #JOB_22_STEP_04;
   END_IF;
END_REGION

REGION Network 110: Step[2204] :
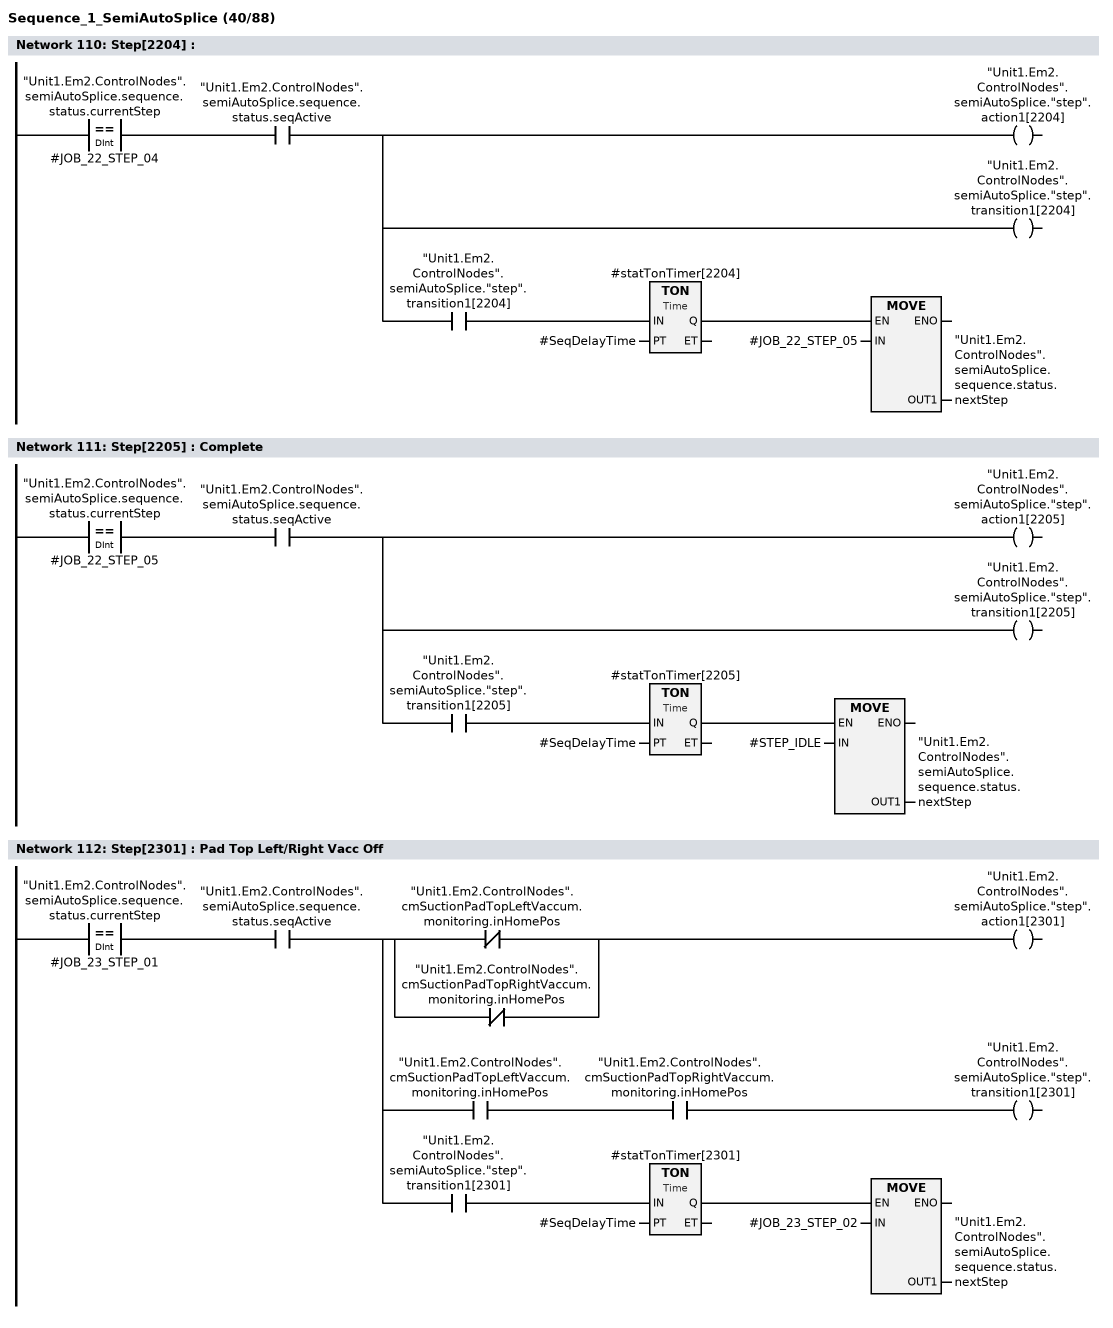
   RUNG wire#powerrail
      { S7_Templates := "SrcType := DInt" } EQ_Contact(in1 := "Unit1.Em2.ControlNodes".semiAutoSplice.sequence.status.currentStep, in2 := #JOB_22_STEP_04)
      Contact( "Unit1.Em2.ControlNodes".semiAutoSplice.sequence.status.seqActive )
      wire#w1
      Coil( "Unit1.Em2.ControlNodes".semiAutoSplice."step".action1[2204] )
   END_RUNG
   RUNG wire#w1
      Coil( "Unit1.Em2.ControlNodes".semiAutoSplice."step".transition1[2204] )
   END_RUNG
   RUNG wire#w1
      Contact( "Unit1.Em2.ControlNodes".semiAutoSplice."step".transition1[2204] )
      { S7_Templates := "time_type := Time" } #statTonTimer[2204].TON(pt := #SeqDelayTime, et =>)
      Move(in := #JOB_22_STEP_05, out1 => "Unit1.Em2.ControlNodes".semiAutoSplice.sequence.status.nextStep)
   END_RUNG
   // the same network as SCL:
   "Unit1.Em2.ControlNodes".semiAutoSplice."step".action1[2204] := ("Unit1.Em2.ControlNodes".semiAutoSplice.sequence.status.currentStep = #JOB_22_STEP_04) AND "Unit1.Em2.ControlNodes".semiAutoSplice.sequence.status.seqActive;
   "Unit1.Em2.ControlNodes".semiAutoSplice."step".transition1[2204] := ("Unit1.Em2.ControlNodes".semiAutoSplice.sequence.status.currentStep = #JOB_22_STEP_04) AND "Unit1.Em2.ControlNodes".semiAutoSplice.sequence.status.seqActive;
   #statTonTimer[2204].TON(IN := ("Unit1.Em2.ControlNodes".semiAutoSplice.sequence.status.currentStep = #JOB_22_STEP_04) AND "Unit1.Em2.ControlNodes".semiAutoSplice.sequence.status.seqActive AND "Unit1.Em2.ControlNodes".semiAutoSplice."step".transition1[2204],
                           PT := #SeqDelayTime);
   IF #statTonTimer[2204].Q THEN
       "Unit1.Em2.ControlNodes".semiAutoSplice.sequence.status.nextStep := #JOB_22_STEP_05;
   END_IF;
END_REGION

REGION Network 111: Step[2205] : Complete
   RUNG wire#powerrail
      { S7_Templates := "SrcType := DInt" } EQ_Contact(in1 := "Unit1.Em2.ControlNodes".semiAutoSplice.sequence.status.currentStep, in2 := #JOB_22_STEP_05)
      Contact( "Unit1.Em2.ControlNodes".semiAutoSplice.sequence.status.seqActive )
      wire#w1
      Coil( "Unit1.Em2.ControlNodes".semiAutoSplice."step".action1[2205] )
   END_RUNG
   RUNG wire#w1
      Coil( "Unit1.Em2.ControlNodes".semiAutoSplice."step".transition1[2205] )
   END_RUNG
   RUNG wire#w1
      Contact( "Unit1.Em2.ControlNodes".semiAutoSplice."step".transition1[2205] )
      { S7_Templates := "time_type := Time" } #statTonTimer[2205].TON(pt := #SeqDelayTime, et =>)
      Move(in := #STEP_IDLE, out1 => "Unit1.Em2.ControlNodes".semiAutoSplice.sequence.status.nextStep)
   END_RUNG
   // the same network as SCL:
   "Unit1.Em2.ControlNodes".semiAutoSplice."step".action1[2205] := ("Unit1.Em2.ControlNodes".semiAutoSplice.sequence.status.currentStep = #JOB_22_STEP_05) AND "Unit1.Em2.ControlNodes".semiAutoSplice.sequence.status.seqActive;
   "Unit1.Em2.ControlNodes".semiAutoSplice."step".transition1[2205] := ("Unit1.Em2.ControlNodes".semiAutoSplice.sequence.status.currentStep = #JOB_22_STEP_05) AND "Unit1.Em2.ControlNodes".semiAutoSplice.sequence.status.seqActive;
   #statTonTimer[2205].TON(IN := ("Unit1.Em2.ControlNodes".semiAutoSplice.sequence.status.currentStep = #JOB_22_STEP_05) AND "Unit1.Em2.ControlNodes".semiAutoSplice.sequence.status.seqActive AND "Unit1.Em2.ControlNodes".semiAutoSplice."step".transition1[2205],
                           PT := #SeqDelayTime);
   IF #statTonTimer[2205].Q THEN
       "Unit1.Em2.ControlNodes".semiAutoSplice.sequence.status.nextStep := #STEP_IDLE;
   END_IF;
END_REGION

REGION Network 112: Step[2301] : Pad Top Left/Right Vacc Off
   RUNG wire#powerrail
      { S7_Templates := "SrcType := DInt" } EQ_Contact(in1 := "Unit1.Em2.ControlNodes".semiAutoSplice.sequence.status.currentStep, in2 := #JOB_23_STEP_01)
      Contact( "Unit1.Em2.ControlNodes".semiAutoSplice.sequence.status.seqActive )
      wire#w1
      I_Contact( "Unit1.Em2.ControlNodes".cmSuctionPadTopLeftVaccum.monitoring.inHomePos )
      wire#w2
      Coil( "Unit1.Em2.ControlNodes".semiAutoSplice."step".action1[2301] )
   END_RUNG
   RUNG wire#w1
      I_Contact( "Unit1.Em2.ControlNodes".cmSuctionPadTopRightVaccum.monitoring.inHomePos )
   END_RUNG wire#w2
   RUNG wire#w1
      Contact( "Unit1.Em2.ControlNodes".cmSuctionPadTopLeftVaccum.monitoring.inHomePos )
      Contact( "Unit1.Em2.ControlNodes".cmSuctionPadTopRightVaccum.monitoring.inHomePos )
      Coil( "Unit1.Em2.ControlNodes".semiAutoSplice."step".transition1[2301] )
   END_RUNG
   RUNG wire#w1
      Contact( "Unit1.Em2.ControlNodes".semiAutoSplice."step".transition1[2301] )
      { S7_Templates := "time_type := Time" } #statTonTimer[2301].TON(pt := #SeqDelayTime, et =>)
      Move(in := #JOB_23_STEP_02, out1 => "Unit1.Em2.ControlNodes".semiAutoSplice.sequence.status.nextStep)
   END_RUNG
   // the same network as SCL:
   #_w1 := ("Unit1.Em2.ControlNodes".semiAutoSplice.sequence.status.currentStep = #JOB_23_STEP_01) AND "Unit1.Em2.ControlNodes".semiAutoSplice.sequence.status.seqActive;
   "Unit1.Em2.ControlNodes".semiAutoSplice."step".action1[2301] := #_w1 AND (NOT "Unit1.Em2.ControlNodes".cmSuctionPadTopLeftVaccum.monitoring.inHomePos OR NOT "Unit1.Em2.ControlNodes".cmSuctionPadTopRightVaccum.monitoring.inHomePos);
   "Unit1.Em2.ControlNodes".semiAutoSplice."step".transition1[2301] := #_w1 AND "Unit1.Em2.ControlNodes".cmSuctionPadTopLeftVaccum.monitoring.inHomePos AND "Unit1.Em2.ControlNodes".cmSuctionPadTopRightVaccum.monitoring.inHomePos;
   #statTonTimer[2301].TON(IN := #_w1 AND "Unit1.Em2.ControlNodes".semiAutoSplice."step".transition1[2301],
                           PT := #SeqDelayTime);
   IF #statTonTimer[2301].Q THEN
       "Unit1.Em2.ControlNodes".semiAutoSplice.sequence.status.nextStep := #JOB_23_STEP_02;
   END_IF;
END_REGION

REGION Network 113: Step[2302] :
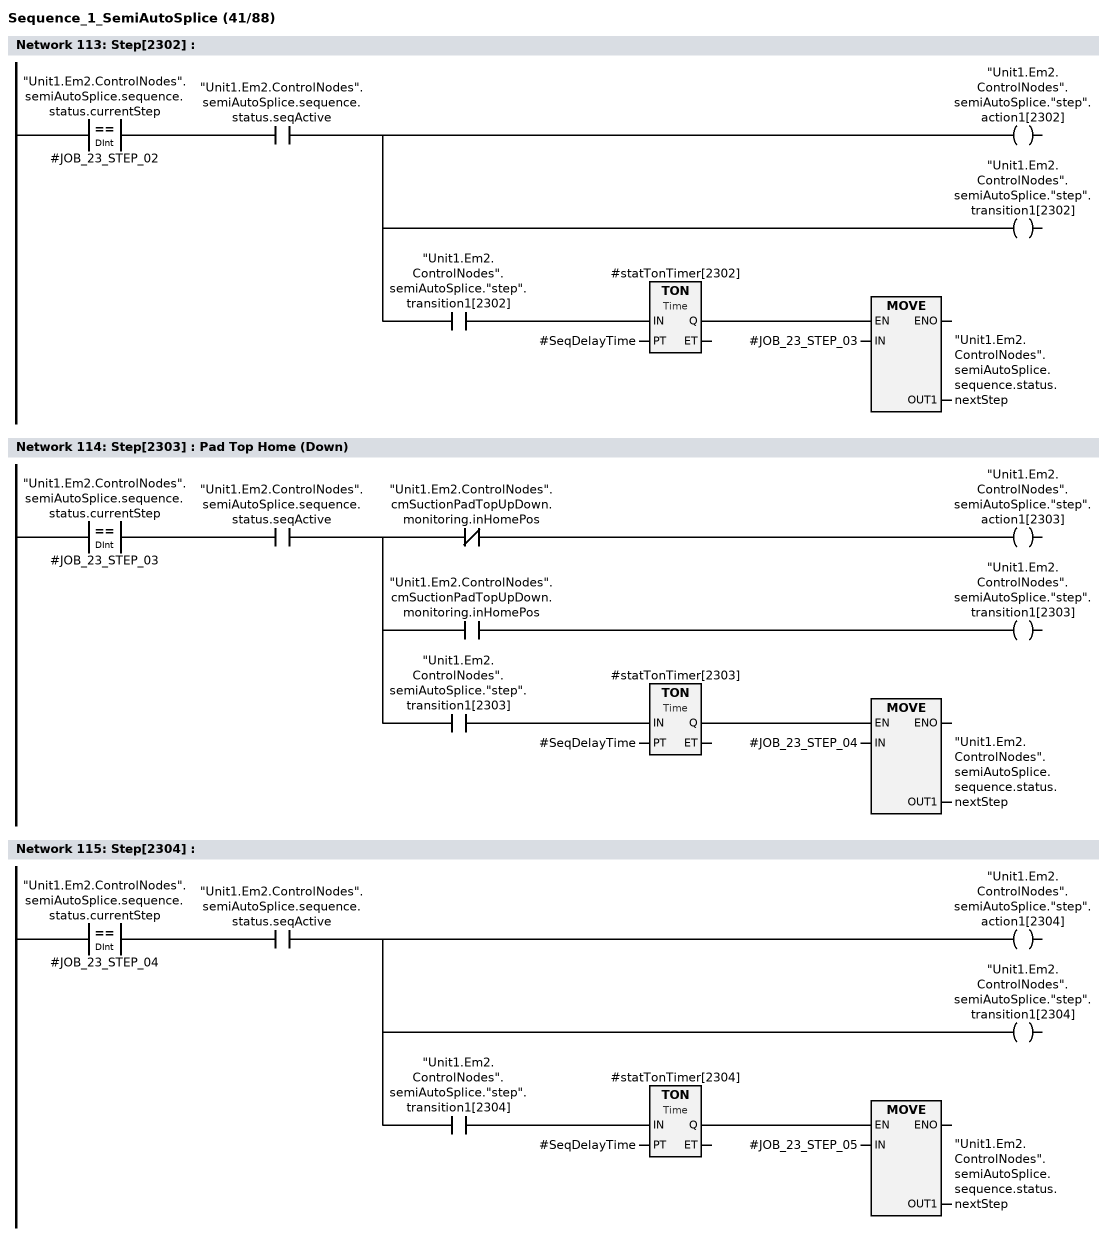
   RUNG wire#powerrail
      { S7_Templates := "SrcType := DInt" } EQ_Contact(in1 := "Unit1.Em2.ControlNodes".semiAutoSplice.sequence.status.currentStep, in2 := #JOB_23_STEP_02)
      Contact( "Unit1.Em2.ControlNodes".semiAutoSplice.sequence.status.seqActive )
      wire#w1
      Coil( "Unit1.Em2.ControlNodes".semiAutoSplice."step".action1[2302] )
   END_RUNG
   RUNG wire#w1
      Coil( "Unit1.Em2.ControlNodes".semiAutoSplice."step".transition1[2302] )
   END_RUNG
   RUNG wire#w1
      Contact( "Unit1.Em2.ControlNodes".semiAutoSplice."step".transition1[2302] )
      { S7_Templates := "time_type := Time" } #statTonTimer[2302].TON(pt := #SeqDelayTime, et =>)
      Move(in := #JOB_23_STEP_03, out1 => "Unit1.Em2.ControlNodes".semiAutoSplice.sequence.status.nextStep)
   END_RUNG
   // the same network as SCL:
   "Unit1.Em2.ControlNodes".semiAutoSplice."step".action1[2302] := ("Unit1.Em2.ControlNodes".semiAutoSplice.sequence.status.currentStep = #JOB_23_STEP_02) AND "Unit1.Em2.ControlNodes".semiAutoSplice.sequence.status.seqActive;
   "Unit1.Em2.ControlNodes".semiAutoSplice."step".transition1[2302] := ("Unit1.Em2.ControlNodes".semiAutoSplice.sequence.status.currentStep = #JOB_23_STEP_02) AND "Unit1.Em2.ControlNodes".semiAutoSplice.sequence.status.seqActive;
   #statTonTimer[2302].TON(IN := ("Unit1.Em2.ControlNodes".semiAutoSplice.sequence.status.currentStep = #JOB_23_STEP_02) AND "Unit1.Em2.ControlNodes".semiAutoSplice.sequence.status.seqActive AND "Unit1.Em2.ControlNodes".semiAutoSplice."step".transition1[2302],
                           PT := #SeqDelayTime);
   IF #statTonTimer[2302].Q THEN
       "Unit1.Em2.ControlNodes".semiAutoSplice.sequence.status.nextStep := #JOB_23_STEP_03;
   END_IF;
END_REGION

REGION Network 114: Step[2303] : Pad Top Home (Down)
   RUNG wire#powerrail
      { S7_Templates := "SrcType := DInt" } EQ_Contact(in1 := "Unit1.Em2.ControlNodes".semiAutoSplice.sequence.status.currentStep, in2 := #JOB_23_STEP_03)
      Contact( "Unit1.Em2.ControlNodes".semiAutoSplice.sequence.status.seqActive )
      wire#w1
      I_Contact( "Unit1.Em2.ControlNodes".cmSuctionPadTopUpDown.monitoring.inHomePos )
      Coil( "Unit1.Em2.ControlNodes".semiAutoSplice."step".action1[2303] )
   END_RUNG
   RUNG wire#w1
      Contact( "Unit1.Em2.ControlNodes".cmSuctionPadTopUpDown.monitoring.inHomePos )
      Coil( "Unit1.Em2.ControlNodes".semiAutoSplice."step".transition1[2303] )
   END_RUNG
   RUNG wire#w1
      Contact( "Unit1.Em2.ControlNodes".semiAutoSplice."step".transition1[2303] )
      { S7_Templates := "time_type := Time" } #statTonTimer[2303].TON(pt := #SeqDelayTime, et =>)
      Move(in := #JOB_23_STEP_04, out1 => "Unit1.Em2.ControlNodes".semiAutoSplice.sequence.status.nextStep)
   END_RUNG
   // the same network as SCL:
   #_w1 := ("Unit1.Em2.ControlNodes".semiAutoSplice.sequence.status.currentStep = #JOB_23_STEP_03) AND "Unit1.Em2.ControlNodes".semiAutoSplice.sequence.status.seqActive;
   "Unit1.Em2.ControlNodes".semiAutoSplice."step".action1[2303] := #_w1 AND NOT "Unit1.Em2.ControlNodes".cmSuctionPadTopUpDown.monitoring.inHomePos;
   "Unit1.Em2.ControlNodes".semiAutoSplice."step".transition1[2303] := #_w1 AND "Unit1.Em2.ControlNodes".cmSuctionPadTopUpDown.monitoring.inHomePos;
   #statTonTimer[2303].TON(IN := #_w1 AND "Unit1.Em2.ControlNodes".semiAutoSplice."step".transition1[2303],
                           PT := #SeqDelayTime);
   IF #statTonTimer[2303].Q THEN
       "Unit1.Em2.ControlNodes".semiAutoSplice.sequence.status.nextStep := #JOB_23_STEP_04;
   END_IF;
END_REGION

REGION Network 115: Step[2304] :
   RUNG wire#powerrail
      { S7_Templates := "SrcType := DInt" } EQ_Contact(in1 := "Unit1.Em2.ControlNodes".semiAutoSplice.sequence.status.currentStep, in2 := #JOB_23_STEP_04)
      Contact( "Unit1.Em2.ControlNodes".semiAutoSplice.sequence.status.seqActive )
      wire#w1
      Coil( "Unit1.Em2.ControlNodes".semiAutoSplice."step".action1[2304] )
   END_RUNG
   RUNG wire#w1
      Coil( "Unit1.Em2.ControlNodes".semiAutoSplice."step".transition1[2304] )
   END_RUNG
   RUNG wire#w1
      Contact( "Unit1.Em2.ControlNodes".semiAutoSplice."step".transition1[2304] )
      { S7_Templates := "time_type := Time" } #statTonTimer[2304].TON(pt := #SeqDelayTime, et =>)
      Move(in := #JOB_23_STEP_05, out1 => "Unit1.Em2.ControlNodes".semiAutoSplice.sequence.status.nextStep)
   END_RUNG
   // the same network as SCL:
   "Unit1.Em2.ControlNodes".semiAutoSplice."step".action1[2304] := ("Unit1.Em2.ControlNodes".semiAutoSplice.sequence.status.currentStep = #JOB_23_STEP_04) AND "Unit1.Em2.ControlNodes".semiAutoSplice.sequence.status.seqActive;
   "Unit1.Em2.ControlNodes".semiAutoSplice."step".transition1[2304] := ("Unit1.Em2.ControlNodes".semiAutoSplice.sequence.status.currentStep = #JOB_23_STEP_04) AND "Unit1.Em2.ControlNodes".semiAutoSplice.sequence.status.seqActive;
   #statTonTimer[2304].TON(IN := ("Unit1.Em2.ControlNodes".semiAutoSplice.sequence.status.currentStep = #JOB_23_STEP_04) AND "Unit1.Em2.ControlNodes".semiAutoSplice.sequence.status.seqActive AND "Unit1.Em2.ControlNodes".semiAutoSplice."step".transition1[2304],
                           PT := #SeqDelayTime);
   IF #statTonTimer[2304].Q THEN
       "Unit1.Em2.ControlNodes".semiAutoSplice.sequence.status.nextStep := #JOB_23_STEP_05;
   END_IF;
END_REGION

REGION Network 116: Step[2305] : Complete
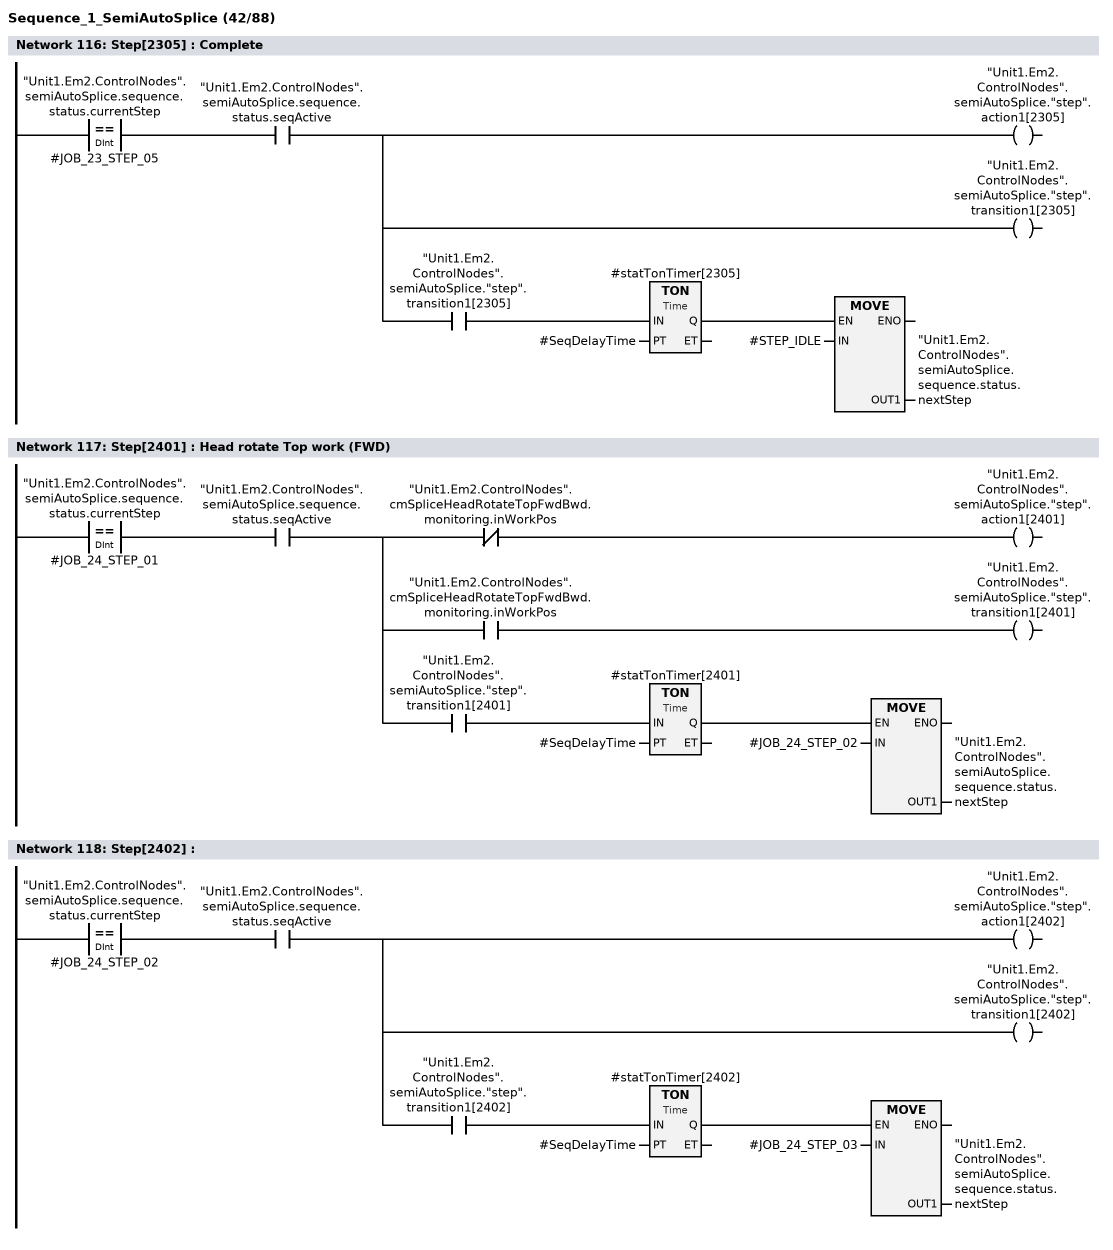
   RUNG wire#powerrail
      { S7_Templates := "SrcType := DInt" } EQ_Contact(in1 := "Unit1.Em2.ControlNodes".semiAutoSplice.sequence.status.currentStep, in2 := #JOB_23_STEP_05)
      Contact( "Unit1.Em2.ControlNodes".semiAutoSplice.sequence.status.seqActive )
      wire#w1
      Coil( "Unit1.Em2.ControlNodes".semiAutoSplice."step".action1[2305] )
   END_RUNG
   RUNG wire#w1
      Coil( "Unit1.Em2.ControlNodes".semiAutoSplice."step".transition1[2305] )
   END_RUNG
   RUNG wire#w1
      Contact( "Unit1.Em2.ControlNodes".semiAutoSplice."step".transition1[2305] )
      { S7_Templates := "time_type := Time" } #statTonTimer[2305].TON(pt := #SeqDelayTime, et =>)
      Move(in := #STEP_IDLE, out1 => "Unit1.Em2.ControlNodes".semiAutoSplice.sequence.status.nextStep)
   END_RUNG
   // the same network as SCL:
   "Unit1.Em2.ControlNodes".semiAutoSplice."step".action1[2305] := ("Unit1.Em2.ControlNodes".semiAutoSplice.sequence.status.currentStep = #JOB_23_STEP_05) AND "Unit1.Em2.ControlNodes".semiAutoSplice.sequence.status.seqActive;
   "Unit1.Em2.ControlNodes".semiAutoSplice."step".transition1[2305] := ("Unit1.Em2.ControlNodes".semiAutoSplice.sequence.status.currentStep = #JOB_23_STEP_05) AND "Unit1.Em2.ControlNodes".semiAutoSplice.sequence.status.seqActive;
   #statTonTimer[2305].TON(IN := ("Unit1.Em2.ControlNodes".semiAutoSplice.sequence.status.currentStep = #JOB_23_STEP_05) AND "Unit1.Em2.ControlNodes".semiAutoSplice.sequence.status.seqActive AND "Unit1.Em2.ControlNodes".semiAutoSplice."step".transition1[2305],
                           PT := #SeqDelayTime);
   IF #statTonTimer[2305].Q THEN
       "Unit1.Em2.ControlNodes".semiAutoSplice.sequence.status.nextStep := #STEP_IDLE;
   END_IF;
END_REGION

REGION Network 117: Step[2401] : Head rotate Top work (FWD)
   RUNG wire#powerrail
      { S7_Templates := "SrcType := DInt" } EQ_Contact(in1 := "Unit1.Em2.ControlNodes".semiAutoSplice.sequence.status.currentStep, in2 := #JOB_24_STEP_01)
      Contact( "Unit1.Em2.ControlNodes".semiAutoSplice.sequence.status.seqActive )
      wire#w1
      I_Contact( "Unit1.Em2.ControlNodes".cmSpliceHeadRotateTopFwdBwd.monitoring.inWorkPos )
      Coil( "Unit1.Em2.ControlNodes".semiAutoSplice."step".action1[2401] )
   END_RUNG
   RUNG wire#w1
      Contact( "Unit1.Em2.ControlNodes".cmSpliceHeadRotateTopFwdBwd.monitoring.inWorkPos )
      Coil( "Unit1.Em2.ControlNodes".semiAutoSplice."step".transition1[2401] )
   END_RUNG
   RUNG wire#w1
      Contact( "Unit1.Em2.ControlNodes".semiAutoSplice."step".transition1[2401] )
      { S7_Templates := "time_type := Time" } #statTonTimer[2401].TON(pt := #SeqDelayTime, et =>)
      Move(in := #JOB_24_STEP_02, out1 => "Unit1.Em2.ControlNodes".semiAutoSplice.sequence.status.nextStep)
   END_RUNG
   // the same network as SCL:
   #_w1 := ("Unit1.Em2.ControlNodes".semiAutoSplice.sequence.status.currentStep = #JOB_24_STEP_01) AND "Unit1.Em2.ControlNodes".semiAutoSplice.sequence.status.seqActive;
   "Unit1.Em2.ControlNodes".semiAutoSplice."step".action1[2401] := #_w1 AND NOT "Unit1.Em2.ControlNodes".cmSpliceHeadRotateTopFwdBwd.monitoring.inWorkPos;
   "Unit1.Em2.ControlNodes".semiAutoSplice."step".transition1[2401] := #_w1 AND "Unit1.Em2.ControlNodes".cmSpliceHeadRotateTopFwdBwd.monitoring.inWorkPos;
   #statTonTimer[2401].TON(IN := #_w1 AND "Unit1.Em2.ControlNodes".semiAutoSplice."step".transition1[2401],
                           PT := #SeqDelayTime);
   IF #statTonTimer[2401].Q THEN
       "Unit1.Em2.ControlNodes".semiAutoSplice.sequence.status.nextStep := #JOB_24_STEP_02;
   END_IF;
END_REGION

REGION Network 118: Step[2402] :
   RUNG wire#powerrail
      { S7_Templates := "SrcType := DInt" } EQ_Contact(in1 := "Unit1.Em2.ControlNodes".semiAutoSplice.sequence.status.currentStep, in2 := #JOB_24_STEP_02)
      Contact( "Unit1.Em2.ControlNodes".semiAutoSplice.sequence.status.seqActive )
      wire#w1
      Coil( "Unit1.Em2.ControlNodes".semiAutoSplice."step".action1[2402] )
   END_RUNG
   RUNG wire#w1
      Coil( "Unit1.Em2.ControlNodes".semiAutoSplice."step".transition1[2402] )
   END_RUNG
   RUNG wire#w1
      Contact( "Unit1.Em2.ControlNodes".semiAutoSplice."step".transition1[2402] )
      { S7_Templates := "time_type := Time" } #statTonTimer[2402].TON(pt := #SeqDelayTime, et =>)
      Move(in := #JOB_24_STEP_03, out1 => "Unit1.Em2.ControlNodes".semiAutoSplice.sequence.status.nextStep)
   END_RUNG
   // the same network as SCL:
   "Unit1.Em2.ControlNodes".semiAutoSplice."step".action1[2402] := ("Unit1.Em2.ControlNodes".semiAutoSplice.sequence.status.currentStep = #JOB_24_STEP_02) AND "Unit1.Em2.ControlNodes".semiAutoSplice.sequence.status.seqActive;
   "Unit1.Em2.ControlNodes".semiAutoSplice."step".transition1[2402] := ("Unit1.Em2.ControlNodes".semiAutoSplice.sequence.status.currentStep = #JOB_24_STEP_02) AND "Unit1.Em2.ControlNodes".semiAutoSplice.sequence.status.seqActive;
   #statTonTimer[2402].TON(IN := ("Unit1.Em2.ControlNodes".semiAutoSplice.sequence.status.currentStep = #JOB_24_STEP_02) AND "Unit1.Em2.ControlNodes".semiAutoSplice.sequence.status.seqActive AND "Unit1.Em2.ControlNodes".semiAutoSplice."step".transition1[2402],
                           PT := #SeqDelayTime);
   IF #statTonTimer[2402].Q THEN
       "Unit1.Em2.ControlNodes".semiAutoSplice.sequence.status.nextStep := #JOB_24_STEP_03;
   END_IF;
END_REGION

REGION Network 119: Step[2403] :
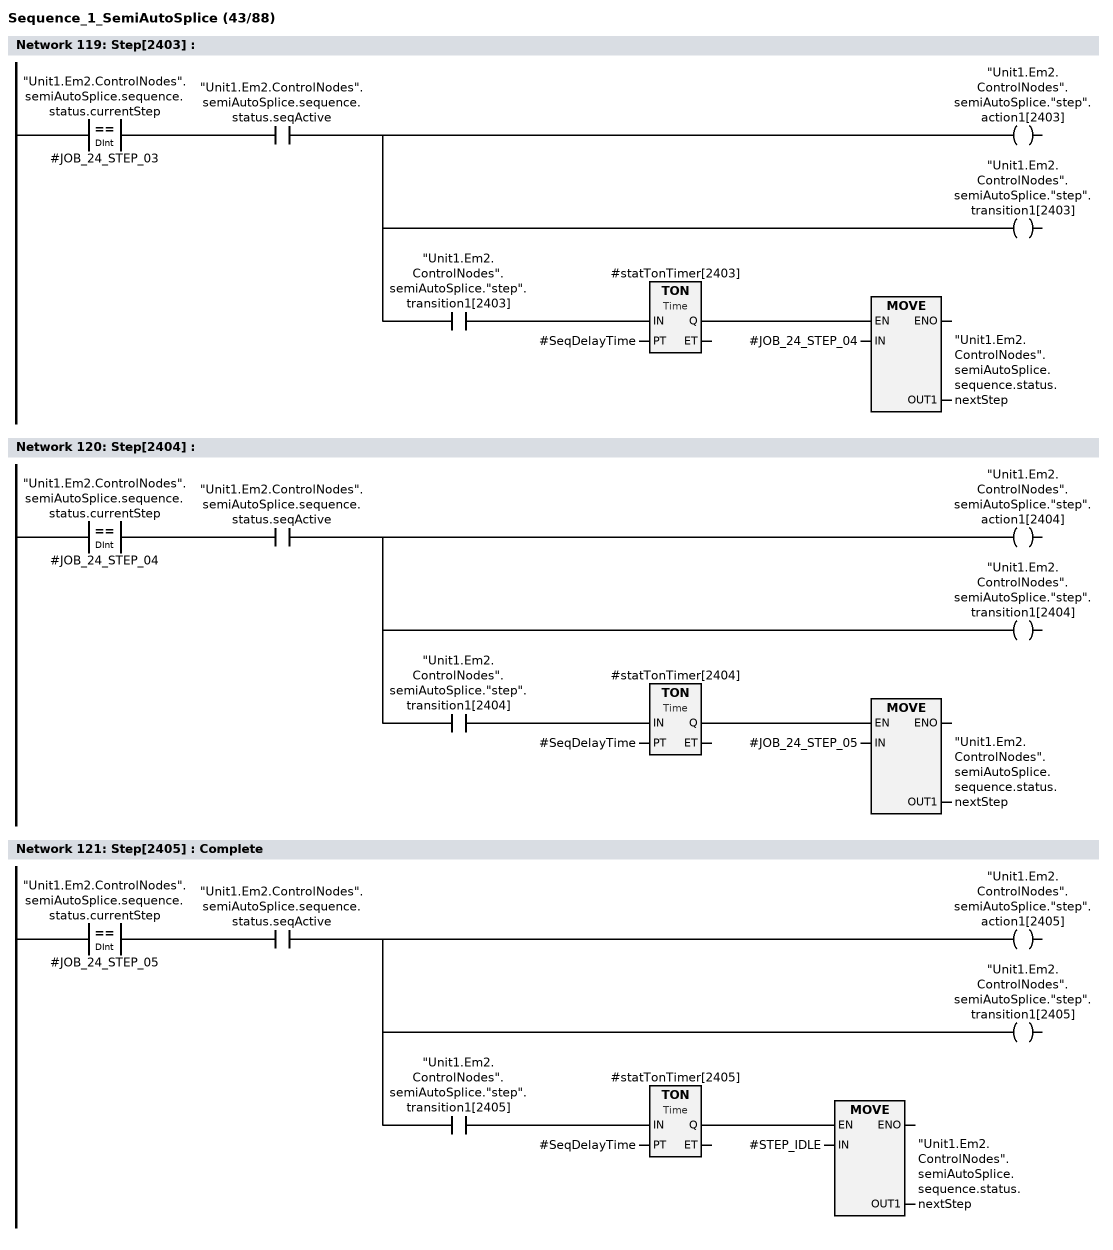
   RUNG wire#powerrail
      { S7_Templates := "SrcType := DInt" } EQ_Contact(in1 := "Unit1.Em2.ControlNodes".semiAutoSplice.sequence.status.currentStep, in2 := #JOB_24_STEP_03)
      Contact( "Unit1.Em2.ControlNodes".semiAutoSplice.sequence.status.seqActive )
      wire#w1
      Coil( "Unit1.Em2.ControlNodes".semiAutoSplice."step".action1[2403] )
   END_RUNG
   RUNG wire#w1
      Coil( "Unit1.Em2.ControlNodes".semiAutoSplice."step".transition1[2403] )
   END_RUNG
   RUNG wire#w1
      Contact( "Unit1.Em2.ControlNodes".semiAutoSplice."step".transition1[2403] )
      { S7_Templates := "time_type := Time" } #statTonTimer[2403].TON(pt := #SeqDelayTime, et =>)
      Move(in := #JOB_24_STEP_04, out1 => "Unit1.Em2.ControlNodes".semiAutoSplice.sequence.status.nextStep)
   END_RUNG
   // the same network as SCL:
   "Unit1.Em2.ControlNodes".semiAutoSplice."step".action1[2403] := ("Unit1.Em2.ControlNodes".semiAutoSplice.sequence.status.currentStep = #JOB_24_STEP_03) AND "Unit1.Em2.ControlNodes".semiAutoSplice.sequence.status.seqActive;
   "Unit1.Em2.ControlNodes".semiAutoSplice."step".transition1[2403] := ("Unit1.Em2.ControlNodes".semiAutoSplice.sequence.status.currentStep = #JOB_24_STEP_03) AND "Unit1.Em2.ControlNodes".semiAutoSplice.sequence.status.seqActive;
   #statTonTimer[2403].TON(IN := ("Unit1.Em2.ControlNodes".semiAutoSplice.sequence.status.currentStep = #JOB_24_STEP_03) AND "Unit1.Em2.ControlNodes".semiAutoSplice.sequence.status.seqActive AND "Unit1.Em2.ControlNodes".semiAutoSplice."step".transition1[2403],
                           PT := #SeqDelayTime);
   IF #statTonTimer[2403].Q THEN
       "Unit1.Em2.ControlNodes".semiAutoSplice.sequence.status.nextStep := #JOB_24_STEP_04;
   END_IF;
END_REGION

REGION Network 120: Step[2404] :
   RUNG wire#powerrail
      { S7_Templates := "SrcType := DInt" } EQ_Contact(in1 := "Unit1.Em2.ControlNodes".semiAutoSplice.sequence.status.currentStep, in2 := #JOB_24_STEP_04)
      Contact( "Unit1.Em2.ControlNodes".semiAutoSplice.sequence.status.seqActive )
      wire#w1
      Coil( "Unit1.Em2.ControlNodes".semiAutoSplice."step".action1[2404] )
   END_RUNG
   RUNG wire#w1
      Coil( "Unit1.Em2.ControlNodes".semiAutoSplice."step".transition1[2404] )
   END_RUNG
   RUNG wire#w1
      Contact( "Unit1.Em2.ControlNodes".semiAutoSplice."step".transition1[2404] )
      { S7_Templates := "time_type := Time" } #statTonTimer[2404].TON(pt := #SeqDelayTime, et =>)
      Move(in := #JOB_24_STEP_05, out1 => "Unit1.Em2.ControlNodes".semiAutoSplice.sequence.status.nextStep)
   END_RUNG
   // the same network as SCL:
   "Unit1.Em2.ControlNodes".semiAutoSplice."step".action1[2404] := ("Unit1.Em2.ControlNodes".semiAutoSplice.sequence.status.currentStep = #JOB_24_STEP_04) AND "Unit1.Em2.ControlNodes".semiAutoSplice.sequence.status.seqActive;
   "Unit1.Em2.ControlNodes".semiAutoSplice."step".transition1[2404] := ("Unit1.Em2.ControlNodes".semiAutoSplice.sequence.status.currentStep = #JOB_24_STEP_04) AND "Unit1.Em2.ControlNodes".semiAutoSplice.sequence.status.seqActive;
   #statTonTimer[2404].TON(IN := ("Unit1.Em2.ControlNodes".semiAutoSplice.sequence.status.currentStep = #JOB_24_STEP_04) AND "Unit1.Em2.ControlNodes".semiAutoSplice.sequence.status.seqActive AND "Unit1.Em2.ControlNodes".semiAutoSplice."step".transition1[2404],
                           PT := #SeqDelayTime);
   IF #statTonTimer[2404].Q THEN
       "Unit1.Em2.ControlNodes".semiAutoSplice.sequence.status.nextStep := #JOB_24_STEP_05;
   END_IF;
END_REGION

REGION Network 121: Step[2405] : Complete
   RUNG wire#powerrail
      { S7_Templates := "SrcType := DInt" } EQ_Contact(in1 := "Unit1.Em2.ControlNodes".semiAutoSplice.sequence.status.currentStep, in2 := #JOB_24_STEP_05)
      Contact( "Unit1.Em2.ControlNodes".semiAutoSplice.sequence.status.seqActive )
      wire#w1
      Coil( "Unit1.Em2.ControlNodes".semiAutoSplice."step".action1[2405] )
   END_RUNG
   RUNG wire#w1
      Coil( "Unit1.Em2.ControlNodes".semiAutoSplice."step".transition1[2405] )
   END_RUNG
   RUNG wire#w1
      Contact( "Unit1.Em2.ControlNodes".semiAutoSplice."step".transition1[2405] )
      { S7_Templates := "time_type := Time" } #statTonTimer[2405].TON(pt := #SeqDelayTime, et =>)
      Move(in := #STEP_IDLE, out1 => "Unit1.Em2.ControlNodes".semiAutoSplice.sequence.status.nextStep)
   END_RUNG
   // the same network as SCL:
   "Unit1.Em2.ControlNodes".semiAutoSplice."step".action1[2405] := ("Unit1.Em2.ControlNodes".semiAutoSplice.sequence.status.currentStep = #JOB_24_STEP_05) AND "Unit1.Em2.ControlNodes".semiAutoSplice.sequence.status.seqActive;
   "Unit1.Em2.ControlNodes".semiAutoSplice."step".transition1[2405] := ("Unit1.Em2.ControlNodes".semiAutoSplice.sequence.status.currentStep = #JOB_24_STEP_05) AND "Unit1.Em2.ControlNodes".semiAutoSplice.sequence.status.seqActive;
   #statTonTimer[2405].TON(IN := ("Unit1.Em2.ControlNodes".semiAutoSplice.sequence.status.currentStep = #JOB_24_STEP_05) AND "Unit1.Em2.ControlNodes".semiAutoSplice.sequence.status.seqActive AND "Unit1.Em2.ControlNodes".semiAutoSplice."step".transition1[2405],
                           PT := #SeqDelayTime);
   IF #statTonTimer[2405].Q THEN
       "Unit1.Em2.ControlNodes".semiAutoSplice.sequence.status.nextStep := #STEP_IDLE;
   END_IF;
END_REGION

REGION Network 122: Step[2501] : Tape Top work (Up)
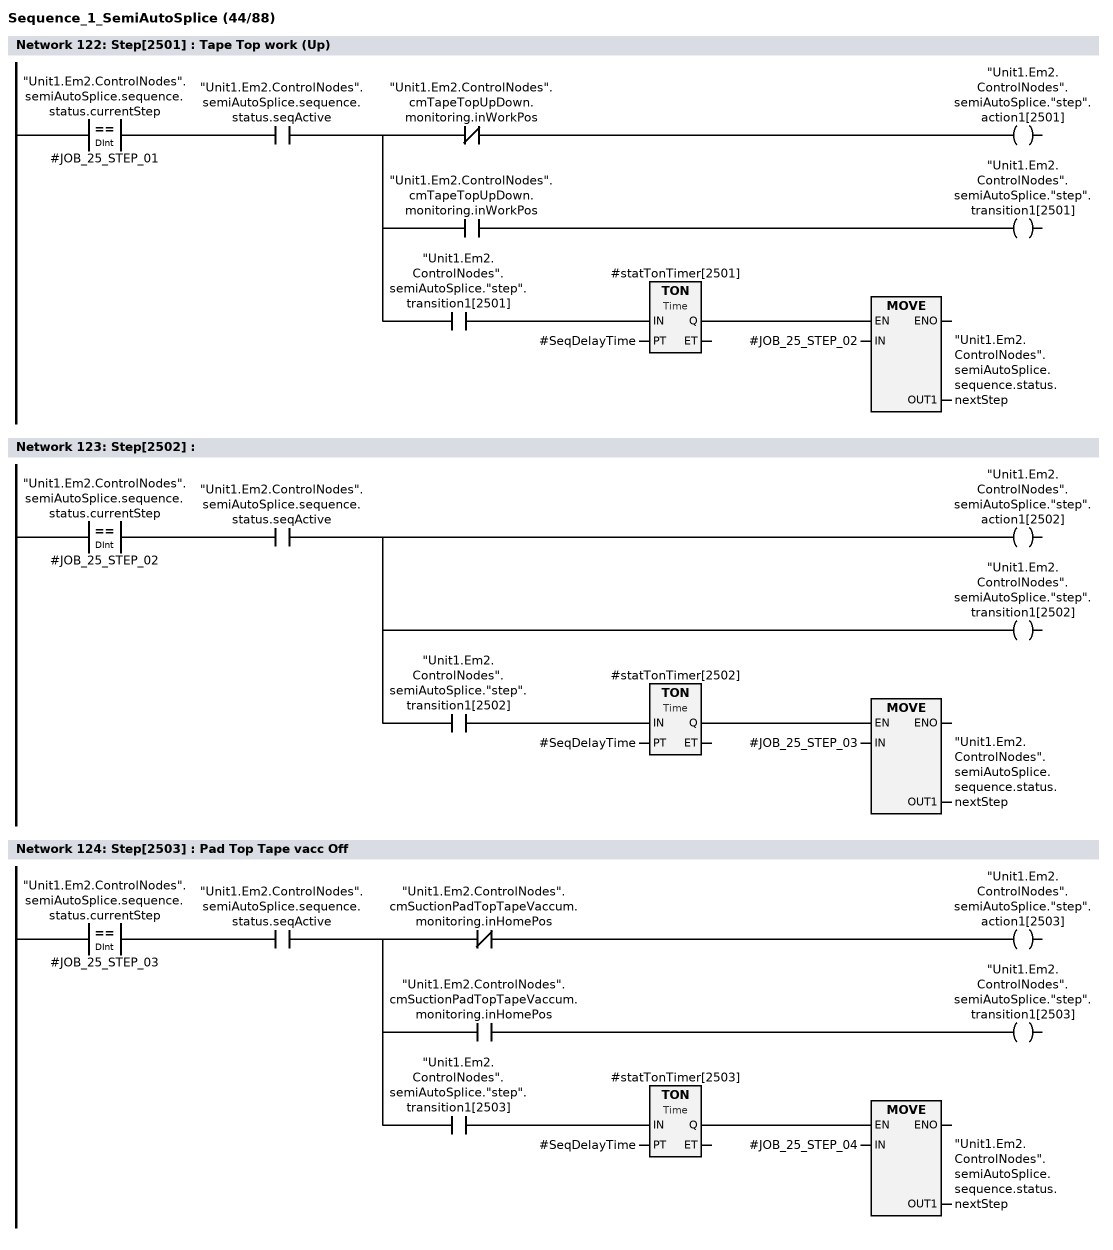
   RUNG wire#powerrail
      { S7_Templates := "SrcType := DInt" } EQ_Contact(in1 := "Unit1.Em2.ControlNodes".semiAutoSplice.sequence.status.currentStep, in2 := #JOB_25_STEP_01)
      Contact( "Unit1.Em2.ControlNodes".semiAutoSplice.sequence.status.seqActive )
      wire#w1
      I_Contact( "Unit1.Em2.ControlNodes".cmTapeTopUpDown.monitoring.inWorkPos )
      Coil( "Unit1.Em2.ControlNodes".semiAutoSplice."step".action1[2501] )
   END_RUNG
   RUNG wire#w1
      Contact( "Unit1.Em2.ControlNodes".cmTapeTopUpDown.monitoring.inWorkPos )
      Coil( "Unit1.Em2.ControlNodes".semiAutoSplice."step".transition1[2501] )
   END_RUNG
   RUNG wire#w1
      Contact( "Unit1.Em2.ControlNodes".semiAutoSplice."step".transition1[2501] )
      { S7_Templates := "time_type := Time" } #statTonTimer[2501].TON(pt := #SeqDelayTime, et =>)
      Move(in := #JOB_25_STEP_02, out1 => "Unit1.Em2.ControlNodes".semiAutoSplice.sequence.status.nextStep)
   END_RUNG
   // the same network as SCL:
   #_w1 := ("Unit1.Em2.ControlNodes".semiAutoSplice.sequence.status.currentStep = #JOB_25_STEP_01) AND "Unit1.Em2.ControlNodes".semiAutoSplice.sequence.status.seqActive;
   "Unit1.Em2.ControlNodes".semiAutoSplice."step".action1[2501] := #_w1 AND NOT "Unit1.Em2.ControlNodes".cmTapeTopUpDown.monitoring.inWorkPos;
   "Unit1.Em2.ControlNodes".semiAutoSplice."step".transition1[2501] := #_w1 AND "Unit1.Em2.ControlNodes".cmTapeTopUpDown.monitoring.inWorkPos;
   #statTonTimer[2501].TON(IN := #_w1 AND "Unit1.Em2.ControlNodes".semiAutoSplice."step".transition1[2501],
                           PT := #SeqDelayTime);
   IF #statTonTimer[2501].Q THEN
       "Unit1.Em2.ControlNodes".semiAutoSplice.sequence.status.nextStep := #JOB_25_STEP_02;
   END_IF;
END_REGION

REGION Network 123: Step[2502] :
   RUNG wire#powerrail
      { S7_Templates := "SrcType := DInt" } EQ_Contact(in1 := "Unit1.Em2.ControlNodes".semiAutoSplice.sequence.status.currentStep, in2 := #JOB_25_STEP_02)
      Contact( "Unit1.Em2.ControlNodes".semiAutoSplice.sequence.status.seqActive )
      wire#w1
      Coil( "Unit1.Em2.ControlNodes".semiAutoSplice."step".action1[2502] )
   END_RUNG
   RUNG wire#w1
      Coil( "Unit1.Em2.ControlNodes".semiAutoSplice."step".transition1[2502] )
   END_RUNG
   RUNG wire#w1
      Contact( "Unit1.Em2.ControlNodes".semiAutoSplice."step".transition1[2502] )
      { S7_Templates := "time_type := Time" } #statTonTimer[2502].TON(pt := #SeqDelayTime, et =>)
      Move(in := #JOB_25_STEP_03, out1 => "Unit1.Em2.ControlNodes".semiAutoSplice.sequence.status.nextStep)
   END_RUNG
   // the same network as SCL:
   "Unit1.Em2.ControlNodes".semiAutoSplice."step".action1[2502] := ("Unit1.Em2.ControlNodes".semiAutoSplice.sequence.status.currentStep = #JOB_25_STEP_02) AND "Unit1.Em2.ControlNodes".semiAutoSplice.sequence.status.seqActive;
   "Unit1.Em2.ControlNodes".semiAutoSplice."step".transition1[2502] := ("Unit1.Em2.ControlNodes".semiAutoSplice.sequence.status.currentStep = #JOB_25_STEP_02) AND "Unit1.Em2.ControlNodes".semiAutoSplice.sequence.status.seqActive;
   #statTonTimer[2502].TON(IN := ("Unit1.Em2.ControlNodes".semiAutoSplice.sequence.status.currentStep = #JOB_25_STEP_02) AND "Unit1.Em2.ControlNodes".semiAutoSplice.sequence.status.seqActive AND "Unit1.Em2.ControlNodes".semiAutoSplice."step".transition1[2502],
                           PT := #SeqDelayTime);
   IF #statTonTimer[2502].Q THEN
       "Unit1.Em2.ControlNodes".semiAutoSplice.sequence.status.nextStep := #JOB_25_STEP_03;
   END_IF;
END_REGION

REGION Network 124: Step[2503] : Pad Top Tape vacc Off
   RUNG wire#powerrail
      { S7_Templates := "SrcType := DInt" } EQ_Contact(in1 := "Unit1.Em2.ControlNodes".semiAutoSplice.sequence.status.currentStep, in2 := #JOB_25_STEP_03)
      Contact( "Unit1.Em2.ControlNodes".semiAutoSplice.sequence.status.seqActive )
      wire#w1
      I_Contact( "Unit1.Em2.ControlNodes".cmSuctionPadTopTapeVaccum.monitoring.inHomePos )
      Coil( "Unit1.Em2.ControlNodes".semiAutoSplice."step".action1[2503] )
   END_RUNG
   RUNG wire#w1
      Contact( "Unit1.Em2.ControlNodes".cmSuctionPadTopTapeVaccum.monitoring.inHomePos )
      Coil( "Unit1.Em2.ControlNodes".semiAutoSplice."step".transition1[2503] )
   END_RUNG
   RUNG wire#w1
      Contact( "Unit1.Em2.ControlNodes".semiAutoSplice."step".transition1[2503] )
      { S7_Templates := "time_type := Time" } #statTonTimer[2503].TON(pt := #SeqDelayTime, et =>)
      Move(in := #JOB_25_STEP_04, out1 => "Unit1.Em2.ControlNodes".semiAutoSplice.sequence.status.nextStep)
   END_RUNG
   // the same network as SCL:
   #_w1 := ("Unit1.Em2.ControlNodes".semiAutoSplice.sequence.status.currentStep = #JOB_25_STEP_03) AND "Unit1.Em2.ControlNodes".semiAutoSplice.sequence.status.seqActive;
   "Unit1.Em2.ControlNodes".semiAutoSplice."step".action1[2503] := #_w1 AND NOT "Unit1.Em2.ControlNodes".cmSuctionPadTopTapeVaccum.monitoring.inHomePos;
   "Unit1.Em2.ControlNodes".semiAutoSplice."step".transition1[2503] := #_w1 AND "Unit1.Em2.ControlNodes".cmSuctionPadTopTapeVaccum.monitoring.inHomePos;
   #statTonTimer[2503].TON(IN := #_w1 AND "Unit1.Em2.ControlNodes".semiAutoSplice."step".transition1[2503],
                           PT := #SeqDelayTime);
   IF #statTonTimer[2503].Q THEN
       "Unit1.Em2.ControlNodes".semiAutoSplice.sequence.status.nextStep := #JOB_25_STEP_04;
   END_IF;
END_REGION

REGION Network 125: Step[2504] :
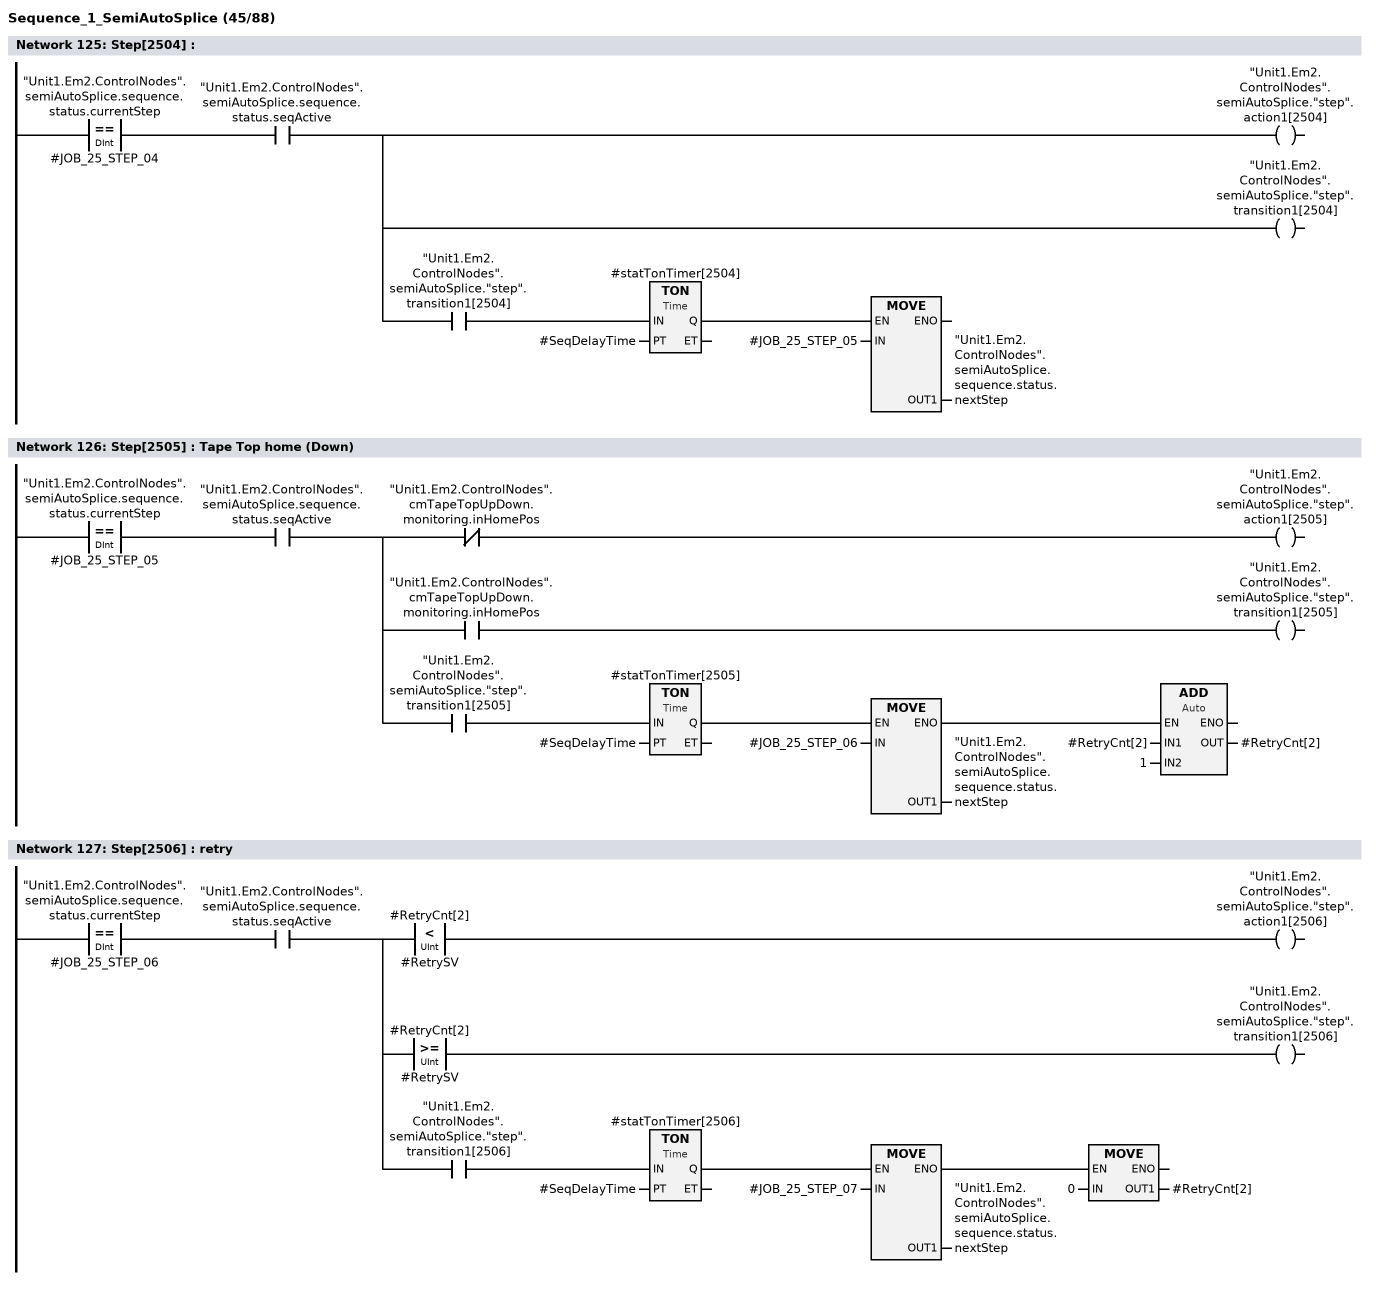
   RUNG wire#powerrail
      { S7_Templates := "SrcType := DInt" } EQ_Contact(in1 := "Unit1.Em2.ControlNodes".semiAutoSplice.sequence.status.currentStep, in2 := #JOB_25_STEP_04)
      Contact( "Unit1.Em2.ControlNodes".semiAutoSplice.sequence.status.seqActive )
      wire#w1
      Coil( "Unit1.Em2.ControlNodes".semiAutoSplice."step".action1[2504] )
   END_RUNG
   RUNG wire#w1
      Coil( "Unit1.Em2.ControlNodes".semiAutoSplice."step".transition1[2504] )
   END_RUNG
   RUNG wire#w1
      Contact( "Unit1.Em2.ControlNodes".semiAutoSplice."step".transition1[2504] )
      { S7_Templates := "time_type := Time" } #statTonTimer[2504].TON(pt := #SeqDelayTime, et =>)
      Move(in := #JOB_25_STEP_05, out1 => "Unit1.Em2.ControlNodes".semiAutoSplice.sequence.status.nextStep)
   END_RUNG
   // the same network as SCL:
   "Unit1.Em2.ControlNodes".semiAutoSplice."step".action1[2504] := ("Unit1.Em2.ControlNodes".semiAutoSplice.sequence.status.currentStep = #JOB_25_STEP_04) AND "Unit1.Em2.ControlNodes".semiAutoSplice.sequence.status.seqActive;
   "Unit1.Em2.ControlNodes".semiAutoSplice."step".transition1[2504] := ("Unit1.Em2.ControlNodes".semiAutoSplice.sequence.status.currentStep = #JOB_25_STEP_04) AND "Unit1.Em2.ControlNodes".semiAutoSplice.sequence.status.seqActive;
   #statTonTimer[2504].TON(IN := ("Unit1.Em2.ControlNodes".semiAutoSplice.sequence.status.currentStep = #JOB_25_STEP_04) AND "Unit1.Em2.ControlNodes".semiAutoSplice.sequence.status.seqActive AND "Unit1.Em2.ControlNodes".semiAutoSplice."step".transition1[2504],
                           PT := #SeqDelayTime);
   IF #statTonTimer[2504].Q THEN
       "Unit1.Em2.ControlNodes".semiAutoSplice.sequence.status.nextStep := #JOB_25_STEP_05;
   END_IF;
END_REGION

REGION Network 126: Step[2505] : Tape Top home (Down)
   RUNG wire#powerrail
      { S7_Templates := "SrcType := DInt" } EQ_Contact(in1 := "Unit1.Em2.ControlNodes".semiAutoSplice.sequence.status.currentStep, in2 := #JOB_25_STEP_05)
      Contact( "Unit1.Em2.ControlNodes".semiAutoSplice.sequence.status.seqActive )
      wire#w1
      I_Contact( "Unit1.Em2.ControlNodes".cmTapeTopUpDown.monitoring.inHomePos )
      Coil( "Unit1.Em2.ControlNodes".semiAutoSplice."step".action1[2505] )
   END_RUNG
   RUNG wire#w1
      Contact( "Unit1.Em2.ControlNodes".cmTapeTopUpDown.monitoring.inHomePos )
      Coil( "Unit1.Em2.ControlNodes".semiAutoSplice."step".transition1[2505] )
   END_RUNG
   RUNG wire#w1
      Contact( "Unit1.Em2.ControlNodes".semiAutoSplice."step".transition1[2505] )
      { S7_Templates := "time_type := Time" } #statTonTimer[2505].TON(pt := #SeqDelayTime, et =>)
      Move(in := #JOB_25_STEP_06, out1 => "Unit1.Em2.ControlNodes".semiAutoSplice.sequence.status.nextStep)
      Add(in1 := #RetryCnt[2], in2 := 1, out => #RetryCnt[2])
   END_RUNG
   // the same network as SCL:
   #_w1 := ("Unit1.Em2.ControlNodes".semiAutoSplice.sequence.status.currentStep = #JOB_25_STEP_05) AND "Unit1.Em2.ControlNodes".semiAutoSplice.sequence.status.seqActive;
   "Unit1.Em2.ControlNodes".semiAutoSplice."step".action1[2505] := #_w1 AND NOT "Unit1.Em2.ControlNodes".cmTapeTopUpDown.monitoring.inHomePos;
   "Unit1.Em2.ControlNodes".semiAutoSplice."step".transition1[2505] := #_w1 AND "Unit1.Em2.ControlNodes".cmTapeTopUpDown.monitoring.inHomePos;
   #statTonTimer[2505].TON(IN := #_w1 AND "Unit1.Em2.ControlNodes".semiAutoSplice."step".transition1[2505],
                           PT := #SeqDelayTime);
   IF #statTonTimer[2505].Q THEN
       "Unit1.Em2.ControlNodes".semiAutoSplice.sequence.status.nextStep := #JOB_25_STEP_06;
       #RetryCnt[2] := #RetryCnt[2] + 1;
   END_IF;
END_REGION

REGION Network 127: Step[2506] : retry
   RUNG wire#powerrail
      { S7_Templates := "SrcType := DInt" } EQ_Contact(in1 := "Unit1.Em2.ControlNodes".semiAutoSplice.sequence.status.currentStep, in2 := #JOB_25_STEP_06)
      Contact( "Unit1.Em2.ControlNodes".semiAutoSplice.sequence.status.seqActive )
      wire#w1
      { S7_Templates := "SrcType := UInt" } LT_Contact(in1 := #RetryCnt[2], in2 := #RetrySV)
      Coil( "Unit1.Em2.ControlNodes".semiAutoSplice."step".action1[2506] )
   END_RUNG
   RUNG wire#w1
      { S7_Templates := "SrcType := UInt" } GE_Contact(in1 := #RetryCnt[2], in2 := #RetrySV)
      Coil( "Unit1.Em2.ControlNodes".semiAutoSplice."step".transition1[2506] )
   END_RUNG
   RUNG wire#w1
      Contact( "Unit1.Em2.ControlNodes".semiAutoSplice."step".transition1[2506] )
      { S7_Templates := "time_type := Time" } #statTonTimer[2506].TON(pt := #SeqDelayTime, et =>)
      Move(in := #JOB_25_STEP_07, out1 => "Unit1.Em2.ControlNodes".semiAutoSplice.sequence.status.nextStep)
      Move(in := 0, out1 => #RetryCnt[2])
   END_RUNG
   // the same network as SCL:
   #_w1 := ("Unit1.Em2.ControlNodes".semiAutoSplice.sequence.status.currentStep = #JOB_25_STEP_06) AND "Unit1.Em2.ControlNodes".semiAutoSplice.sequence.status.seqActive;
   "Unit1.Em2.ControlNodes".semiAutoSplice."step".action1[2506] := #_w1 AND (#RetryCnt[2] < #RetrySV);
   "Unit1.Em2.ControlNodes".semiAutoSplice."step".transition1[2506] := #_w1 AND (#RetryCnt[2] >= #RetrySV);
   #statTonTimer[2506].TON(IN := #_w1 AND "Unit1.Em2.ControlNodes".semiAutoSplice."step".transition1[2506],
                           PT := #SeqDelayTime);
   IF #statTonTimer[2506].Q THEN
       "Unit1.Em2.ControlNodes".semiAutoSplice.sequence.status.nextStep := #JOB_25_STEP_07;
       #RetryCnt[2] := 0;
   END_IF;
END_REGION

REGION Network 128: Step[2507] : Complete
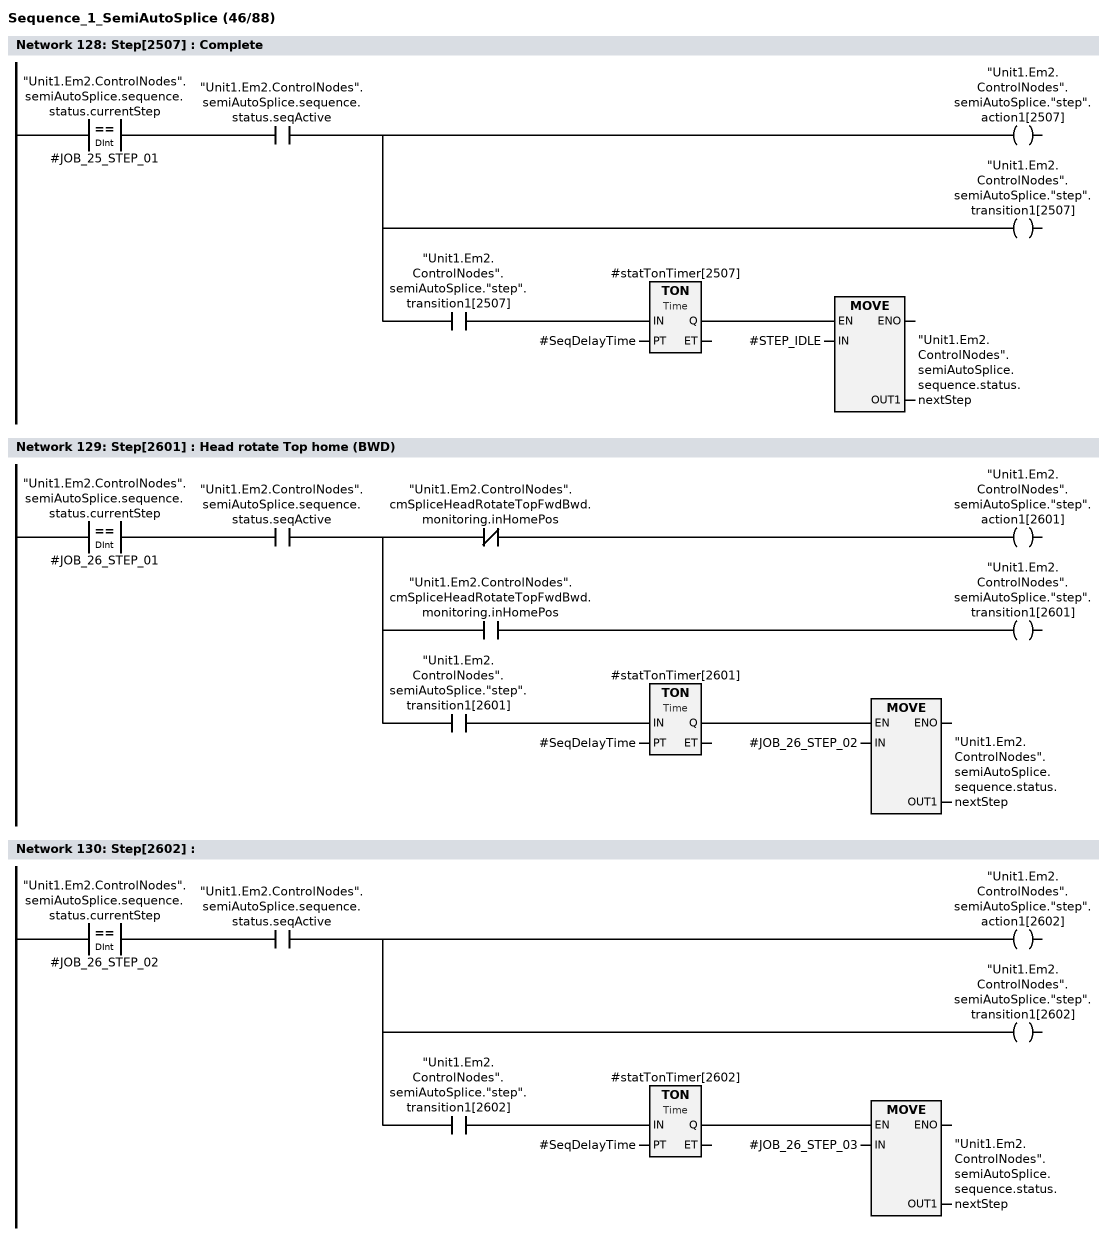
   RUNG wire#powerrail
      { S7_Templates := "SrcType := DInt" } EQ_Contact(in1 := "Unit1.Em2.ControlNodes".semiAutoSplice.sequence.status.currentStep, in2 := #JOB_25_STEP_01)
      Contact( "Unit1.Em2.ControlNodes".semiAutoSplice.sequence.status.seqActive )
      wire#w1
      Coil( "Unit1.Em2.ControlNodes".semiAutoSplice."step".action1[2507] )
   END_RUNG
   RUNG wire#w1
      Coil( "Unit1.Em2.ControlNodes".semiAutoSplice."step".transition1[2507] )
   END_RUNG
   RUNG wire#w1
      Contact( "Unit1.Em2.ControlNodes".semiAutoSplice."step".transition1[2507] )
      { S7_Templates := "time_type := Time" } #statTonTimer[2507].TON(pt := #SeqDelayTime, et =>)
      Move(in := #STEP_IDLE, out1 => "Unit1.Em2.ControlNodes".semiAutoSplice.sequence.status.nextStep)
   END_RUNG
   // the same network as SCL:
   "Unit1.Em2.ControlNodes".semiAutoSplice."step".action1[2507] := ("Unit1.Em2.ControlNodes".semiAutoSplice.sequence.status.currentStep = #JOB_25_STEP_01) AND "Unit1.Em2.ControlNodes".semiAutoSplice.sequence.status.seqActive;
   "Unit1.Em2.ControlNodes".semiAutoSplice."step".transition1[2507] := ("Unit1.Em2.ControlNodes".semiAutoSplice.sequence.status.currentStep = #JOB_25_STEP_01) AND "Unit1.Em2.ControlNodes".semiAutoSplice.sequence.status.seqActive;
   #statTonTimer[2507].TON(IN := ("Unit1.Em2.ControlNodes".semiAutoSplice.sequence.status.currentStep = #JOB_25_STEP_01) AND "Unit1.Em2.ControlNodes".semiAutoSplice.sequence.status.seqActive AND "Unit1.Em2.ControlNodes".semiAutoSplice."step".transition1[2507],
                           PT := #SeqDelayTime);
   IF #statTonTimer[2507].Q THEN
       "Unit1.Em2.ControlNodes".semiAutoSplice.sequence.status.nextStep := #STEP_IDLE;
   END_IF;
END_REGION

REGION Network 129: Step[2601] : Head rotate Top home (BWD)
   RUNG wire#powerrail
      { S7_Templates := "SrcType := DInt" } EQ_Contact(in1 := "Unit1.Em2.ControlNodes".semiAutoSplice.sequence.status.currentStep, in2 := #JOB_26_STEP_01)
      Contact( "Unit1.Em2.ControlNodes".semiAutoSplice.sequence.status.seqActive )
      wire#w1
      I_Contact( "Unit1.Em2.ControlNodes".cmSpliceHeadRotateTopFwdBwd.monitoring.inHomePos )
      Coil( "Unit1.Em2.ControlNodes".semiAutoSplice."step".action1[2601] )
   END_RUNG
   RUNG wire#w1
      Contact( "Unit1.Em2.ControlNodes".cmSpliceHeadRotateTopFwdBwd.monitoring.inHomePos )
      Coil( "Unit1.Em2.ControlNodes".semiAutoSplice."step".transition1[2601] )
   END_RUNG
   RUNG wire#w1
      Contact( "Unit1.Em2.ControlNodes".semiAutoSplice."step".transition1[2601] )
      { S7_Templates := "time_type := Time" } #statTonTimer[2601].TON(pt := #SeqDelayTime, et =>)
      Move(in := #JOB_26_STEP_02, out1 => "Unit1.Em2.ControlNodes".semiAutoSplice.sequence.status.nextStep)
   END_RUNG
   // the same network as SCL:
   #_w1 := ("Unit1.Em2.ControlNodes".semiAutoSplice.sequence.status.currentStep = #JOB_26_STEP_01) AND "Unit1.Em2.ControlNodes".semiAutoSplice.sequence.status.seqActive;
   "Unit1.Em2.ControlNodes".semiAutoSplice."step".action1[2601] := #_w1 AND NOT "Unit1.Em2.ControlNodes".cmSpliceHeadRotateTopFwdBwd.monitoring.inHomePos;
   "Unit1.Em2.ControlNodes".semiAutoSplice."step".transition1[2601] := #_w1 AND "Unit1.Em2.ControlNodes".cmSpliceHeadRotateTopFwdBwd.monitoring.inHomePos;
   #statTonTimer[2601].TON(IN := #_w1 AND "Unit1.Em2.ControlNodes".semiAutoSplice."step".transition1[2601],
                           PT := #SeqDelayTime);
   IF #statTonTimer[2601].Q THEN
       "Unit1.Em2.ControlNodes".semiAutoSplice.sequence.status.nextStep := #JOB_26_STEP_02;
   END_IF;
END_REGION

REGION Network 130: Step[2602] :
   RUNG wire#powerrail
      { S7_Templates := "SrcType := DInt" } EQ_Contact(in1 := "Unit1.Em2.ControlNodes".semiAutoSplice.sequence.status.currentStep, in2 := #JOB_26_STEP_02)
      Contact( "Unit1.Em2.ControlNodes".semiAutoSplice.sequence.status.seqActive )
      wire#w1
      Coil( "Unit1.Em2.ControlNodes".semiAutoSplice."step".action1[2602] )
   END_RUNG
   RUNG wire#w1
      Coil( "Unit1.Em2.ControlNodes".semiAutoSplice."step".transition1[2602] )
   END_RUNG
   RUNG wire#w1
      Contact( "Unit1.Em2.ControlNodes".semiAutoSplice."step".transition1[2602] )
      { S7_Templates := "time_type := Time" } #statTonTimer[2602].TON(pt := #SeqDelayTime, et =>)
      Move(in := #JOB_26_STEP_03, out1 => "Unit1.Em2.ControlNodes".semiAutoSplice.sequence.status.nextStep)
   END_RUNG
   // the same network as SCL:
   "Unit1.Em2.ControlNodes".semiAutoSplice."step".action1[2602] := ("Unit1.Em2.ControlNodes".semiAutoSplice.sequence.status.currentStep = #JOB_26_STEP_02) AND "Unit1.Em2.ControlNodes".semiAutoSplice.sequence.status.seqActive;
   "Unit1.Em2.ControlNodes".semiAutoSplice."step".transition1[2602] := ("Unit1.Em2.ControlNodes".semiAutoSplice.sequence.status.currentStep = #JOB_26_STEP_02) AND "Unit1.Em2.ControlNodes".semiAutoSplice.sequence.status.seqActive;
   #statTonTimer[2602].TON(IN := ("Unit1.Em2.ControlNodes".semiAutoSplice.sequence.status.currentStep = #JOB_26_STEP_02) AND "Unit1.Em2.ControlNodes".semiAutoSplice.sequence.status.seqActive AND "Unit1.Em2.ControlNodes".semiAutoSplice."step".transition1[2602],
                           PT := #SeqDelayTime);
   IF #statTonTimer[2602].Q THEN
       "Unit1.Em2.ControlNodes".semiAutoSplice.sequence.status.nextStep := #JOB_26_STEP_03;
   END_IF;
END_REGION

REGION Network 131: Step[2603] :
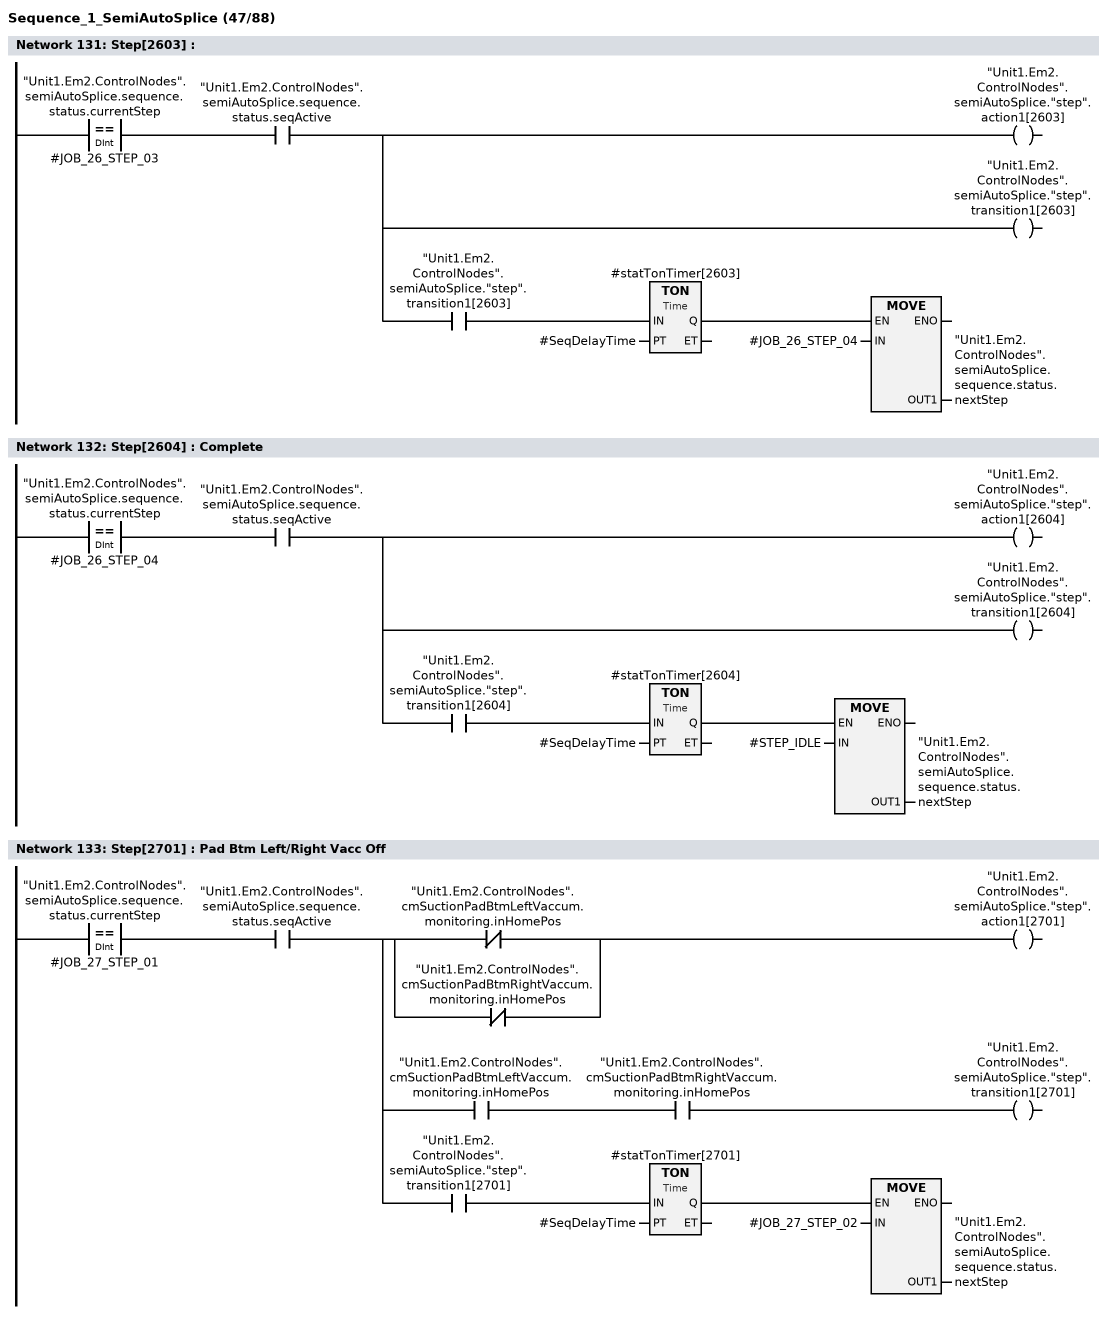
   RUNG wire#powerrail
      { S7_Templates := "SrcType := DInt" } EQ_Contact(in1 := "Unit1.Em2.ControlNodes".semiAutoSplice.sequence.status.currentStep, in2 := #JOB_26_STEP_03)
      Contact( "Unit1.Em2.ControlNodes".semiAutoSplice.sequence.status.seqActive )
      wire#w1
      Coil( "Unit1.Em2.ControlNodes".semiAutoSplice."step".action1[2603] )
   END_RUNG
   RUNG wire#w1
      Coil( "Unit1.Em2.ControlNodes".semiAutoSplice."step".transition1[2603] )
   END_RUNG
   RUNG wire#w1
      Contact( "Unit1.Em2.ControlNodes".semiAutoSplice."step".transition1[2603] )
      { S7_Templates := "time_type := Time" } #statTonTimer[2603].TON(pt := #SeqDelayTime, et =>)
      Move(in := #JOB_26_STEP_04, out1 => "Unit1.Em2.ControlNodes".semiAutoSplice.sequence.status.nextStep)
   END_RUNG
   // the same network as SCL:
   "Unit1.Em2.ControlNodes".semiAutoSplice."step".action1[2603] := ("Unit1.Em2.ControlNodes".semiAutoSplice.sequence.status.currentStep = #JOB_26_STEP_03) AND "Unit1.Em2.ControlNodes".semiAutoSplice.sequence.status.seqActive;
   "Unit1.Em2.ControlNodes".semiAutoSplice."step".transition1[2603] := ("Unit1.Em2.ControlNodes".semiAutoSplice.sequence.status.currentStep = #JOB_26_STEP_03) AND "Unit1.Em2.ControlNodes".semiAutoSplice.sequence.status.seqActive;
   #statTonTimer[2603].TON(IN := ("Unit1.Em2.ControlNodes".semiAutoSplice.sequence.status.currentStep = #JOB_26_STEP_03) AND "Unit1.Em2.ControlNodes".semiAutoSplice.sequence.status.seqActive AND "Unit1.Em2.ControlNodes".semiAutoSplice."step".transition1[2603],
                           PT := #SeqDelayTime);
   IF #statTonTimer[2603].Q THEN
       "Unit1.Em2.ControlNodes".semiAutoSplice.sequence.status.nextStep := #JOB_26_STEP_04;
   END_IF;
END_REGION

REGION Network 132: Step[2604] : Complete
   RUNG wire#powerrail
      { S7_Templates := "SrcType := DInt" } EQ_Contact(in1 := "Unit1.Em2.ControlNodes".semiAutoSplice.sequence.status.currentStep, in2 := #JOB_26_STEP_04)
      Contact( "Unit1.Em2.ControlNodes".semiAutoSplice.sequence.status.seqActive )
      wire#w1
      Coil( "Unit1.Em2.ControlNodes".semiAutoSplice."step".action1[2604] )
   END_RUNG
   RUNG wire#w1
      Coil( "Unit1.Em2.ControlNodes".semiAutoSplice."step".transition1[2604] )
   END_RUNG
   RUNG wire#w1
      Contact( "Unit1.Em2.ControlNodes".semiAutoSplice."step".transition1[2604] )
      { S7_Templates := "time_type := Time" } #statTonTimer[2604].TON(pt := #SeqDelayTime, et =>)
      Move(in := #STEP_IDLE, out1 => "Unit1.Em2.ControlNodes".semiAutoSplice.sequence.status.nextStep)
   END_RUNG
   // the same network as SCL:
   "Unit1.Em2.ControlNodes".semiAutoSplice."step".action1[2604] := ("Unit1.Em2.ControlNodes".semiAutoSplice.sequence.status.currentStep = #JOB_26_STEP_04) AND "Unit1.Em2.ControlNodes".semiAutoSplice.sequence.status.seqActive;
   "Unit1.Em2.ControlNodes".semiAutoSplice."step".transition1[2604] := ("Unit1.Em2.ControlNodes".semiAutoSplice.sequence.status.currentStep = #JOB_26_STEP_04) AND "Unit1.Em2.ControlNodes".semiAutoSplice.sequence.status.seqActive;
   #statTonTimer[2604].TON(IN := ("Unit1.Em2.ControlNodes".semiAutoSplice.sequence.status.currentStep = #JOB_26_STEP_04) AND "Unit1.Em2.ControlNodes".semiAutoSplice.sequence.status.seqActive AND "Unit1.Em2.ControlNodes".semiAutoSplice."step".transition1[2604],
                           PT := #SeqDelayTime);
   IF #statTonTimer[2604].Q THEN
       "Unit1.Em2.ControlNodes".semiAutoSplice.sequence.status.nextStep := #STEP_IDLE;
   END_IF;
END_REGION

REGION Network 133: Step[2701] : Pad Btm Left/Right Vacc Off
   RUNG wire#powerrail
      { S7_Templates := "SrcType := DInt" } EQ_Contact(in1 := "Unit1.Em2.ControlNodes".semiAutoSplice.sequence.status.currentStep, in2 := #JOB_27_STEP_01)
      Contact( "Unit1.Em2.ControlNodes".semiAutoSplice.sequence.status.seqActive )
      wire#w1
      I_Contact( "Unit1.Em2.ControlNodes".cmSuctionPadBtmLeftVaccum.monitoring.inHomePos )
      wire#w2
      Coil( "Unit1.Em2.ControlNodes".semiAutoSplice."step".action1[2701] )
   END_RUNG
   RUNG wire#w1
      I_Contact( "Unit1.Em2.ControlNodes".cmSuctionPadBtmRightVaccum.monitoring.inHomePos )
   END_RUNG wire#w2
   RUNG wire#w1
      Contact( "Unit1.Em2.ControlNodes".cmSuctionPadBtmLeftVaccum.monitoring.inHomePos )
      Contact( "Unit1.Em2.ControlNodes".cmSuctionPadBtmRightVaccum.monitoring.inHomePos )
      Coil( "Unit1.Em2.ControlNodes".semiAutoSplice."step".transition1[2701] )
   END_RUNG
   RUNG wire#w1
      Contact( "Unit1.Em2.ControlNodes".semiAutoSplice."step".transition1[2701] )
      { S7_Templates := "time_type := Time" } #statTonTimer[2701].TON(pt := #SeqDelayTime, et =>)
      Move(in := #JOB_27_STEP_02, out1 => "Unit1.Em2.ControlNodes".semiAutoSplice.sequence.status.nextStep)
   END_RUNG
   // the same network as SCL:
   #_w1 := ("Unit1.Em2.ControlNodes".semiAutoSplice.sequence.status.currentStep = #JOB_27_STEP_01) AND "Unit1.Em2.ControlNodes".semiAutoSplice.sequence.status.seqActive;
   "Unit1.Em2.ControlNodes".semiAutoSplice."step".action1[2701] := #_w1 AND (NOT "Unit1.Em2.ControlNodes".cmSuctionPadBtmLeftVaccum.monitoring.inHomePos OR NOT "Unit1.Em2.ControlNodes".cmSuctionPadBtmRightVaccum.monitoring.inHomePos);
   "Unit1.Em2.ControlNodes".semiAutoSplice."step".transition1[2701] := #_w1 AND "Unit1.Em2.ControlNodes".cmSuctionPadBtmLeftVaccum.monitoring.inHomePos AND "Unit1.Em2.ControlNodes".cmSuctionPadBtmRightVaccum.monitoring.inHomePos;
   #statTonTimer[2701].TON(IN := #_w1 AND "Unit1.Em2.ControlNodes".semiAutoSplice."step".transition1[2701],
                           PT := #SeqDelayTime);
   IF #statTonTimer[2701].Q THEN
       "Unit1.Em2.ControlNodes".semiAutoSplice.sequence.status.nextStep := #JOB_27_STEP_02;
   END_IF;
END_REGION

REGION Network 134: Step[2702] :
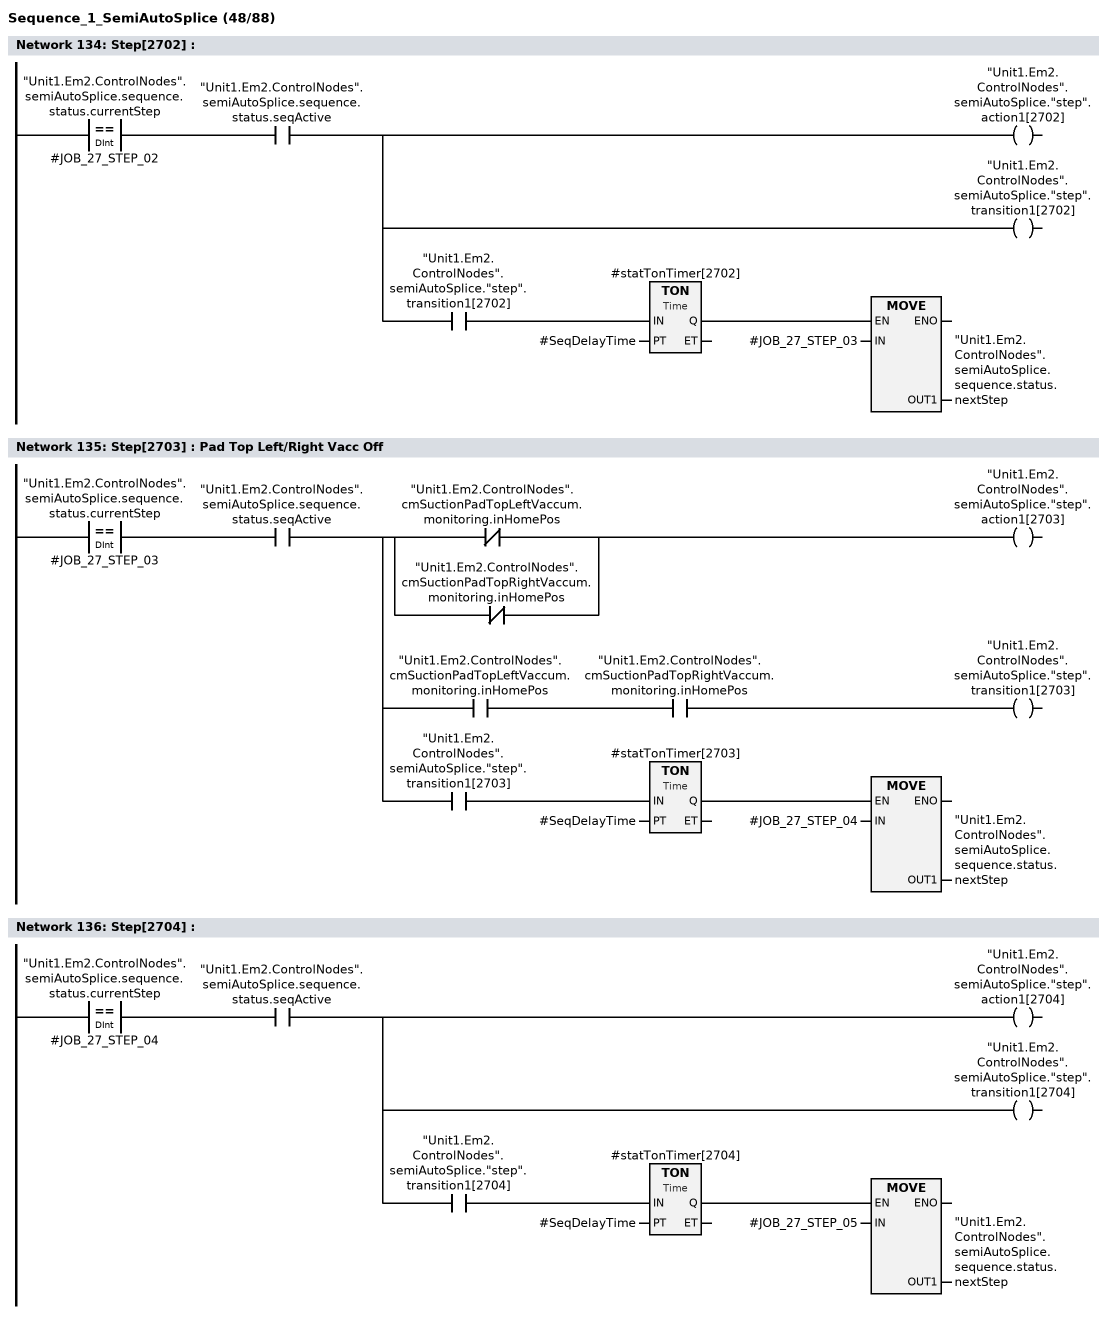
   RUNG wire#powerrail
      { S7_Templates := "SrcType := DInt" } EQ_Contact(in1 := "Unit1.Em2.ControlNodes".semiAutoSplice.sequence.status.currentStep, in2 := #JOB_27_STEP_02)
      Contact( "Unit1.Em2.ControlNodes".semiAutoSplice.sequence.status.seqActive )
      wire#w1
      Coil( "Unit1.Em2.ControlNodes".semiAutoSplice."step".action1[2702] )
   END_RUNG
   RUNG wire#w1
      Coil( "Unit1.Em2.ControlNodes".semiAutoSplice."step".transition1[2702] )
   END_RUNG
   RUNG wire#w1
      Contact( "Unit1.Em2.ControlNodes".semiAutoSplice."step".transition1[2702] )
      { S7_Templates := "time_type := Time" } #statTonTimer[2702].TON(pt := #SeqDelayTime, et =>)
      Move(in := #JOB_27_STEP_03, out1 => "Unit1.Em2.ControlNodes".semiAutoSplice.sequence.status.nextStep)
   END_RUNG
   // the same network as SCL:
   "Unit1.Em2.ControlNodes".semiAutoSplice."step".action1[2702] := ("Unit1.Em2.ControlNodes".semiAutoSplice.sequence.status.currentStep = #JOB_27_STEP_02) AND "Unit1.Em2.ControlNodes".semiAutoSplice.sequence.status.seqActive;
   "Unit1.Em2.ControlNodes".semiAutoSplice."step".transition1[2702] := ("Unit1.Em2.ControlNodes".semiAutoSplice.sequence.status.currentStep = #JOB_27_STEP_02) AND "Unit1.Em2.ControlNodes".semiAutoSplice.sequence.status.seqActive;
   #statTonTimer[2702].TON(IN := ("Unit1.Em2.ControlNodes".semiAutoSplice.sequence.status.currentStep = #JOB_27_STEP_02) AND "Unit1.Em2.ControlNodes".semiAutoSplice.sequence.status.seqActive AND "Unit1.Em2.ControlNodes".semiAutoSplice."step".transition1[2702],
                           PT := #SeqDelayTime);
   IF #statTonTimer[2702].Q THEN
       "Unit1.Em2.ControlNodes".semiAutoSplice.sequence.status.nextStep := #JOB_27_STEP_03;
   END_IF;
END_REGION

REGION Network 135: Step[2703] : Pad Top Left/Right Vacc Off
   RUNG wire#powerrail
      { S7_Templates := "SrcType := DInt" } EQ_Contact(in1 := "Unit1.Em2.ControlNodes".semiAutoSplice.sequence.status.currentStep, in2 := #JOB_27_STEP_03)
      Contact( "Unit1.Em2.ControlNodes".semiAutoSplice.sequence.status.seqActive )
      wire#w1
      I_Contact( "Unit1.Em2.ControlNodes".cmSuctionPadTopLeftVaccum.monitoring.inHomePos )
      wire#w2
      Coil( "Unit1.Em2.ControlNodes".semiAutoSplice."step".action1[2703] )
   END_RUNG
   RUNG wire#w1
      I_Contact( "Unit1.Em2.ControlNodes".cmSuctionPadTopRightVaccum.monitoring.inHomePos )
   END_RUNG wire#w2
   RUNG wire#w1
      Contact( "Unit1.Em2.ControlNodes".cmSuctionPadTopLeftVaccum.monitoring.inHomePos )
      Contact( "Unit1.Em2.ControlNodes".cmSuctionPadTopRightVaccum.monitoring.inHomePos )
      Coil( "Unit1.Em2.ControlNodes".semiAutoSplice."step".transition1[2703] )
   END_RUNG
   RUNG wire#w1
      Contact( "Unit1.Em2.ControlNodes".semiAutoSplice."step".transition1[2703] )
      { S7_Templates := "time_type := Time" } #statTonTimer[2703].TON(pt := #SeqDelayTime, et =>)
      Move(in := #JOB_27_STEP_04, out1 => "Unit1.Em2.ControlNodes".semiAutoSplice.sequence.status.nextStep)
   END_RUNG
   // the same network as SCL:
   #_w1 := ("Unit1.Em2.ControlNodes".semiAutoSplice.sequence.status.currentStep = #JOB_27_STEP_03) AND "Unit1.Em2.ControlNodes".semiAutoSplice.sequence.status.seqActive;
   "Unit1.Em2.ControlNodes".semiAutoSplice."step".action1[2703] := #_w1 AND (NOT "Unit1.Em2.ControlNodes".cmSuctionPadTopLeftVaccum.monitoring.inHomePos OR NOT "Unit1.Em2.ControlNodes".cmSuctionPadTopRightVaccum.monitoring.inHomePos);
   "Unit1.Em2.ControlNodes".semiAutoSplice."step".transition1[2703] := #_w1 AND "Unit1.Em2.ControlNodes".cmSuctionPadTopLeftVaccum.monitoring.inHomePos AND "Unit1.Em2.ControlNodes".cmSuctionPadTopRightVaccum.monitoring.inHomePos;
   #statTonTimer[2703].TON(IN := #_w1 AND "Unit1.Em2.ControlNodes".semiAutoSplice."step".transition1[2703],
                           PT := #SeqDelayTime);
   IF #statTonTimer[2703].Q THEN
       "Unit1.Em2.ControlNodes".semiAutoSplice.sequence.status.nextStep := #JOB_27_STEP_04;
   END_IF;
END_REGION

REGION Network 136: Step[2704] :
   RUNG wire#powerrail
      { S7_Templates := "SrcType := DInt" } EQ_Contact(in1 := "Unit1.Em2.ControlNodes".semiAutoSplice.sequence.status.currentStep, in2 := #JOB_27_STEP_04)
      Contact( "Unit1.Em2.ControlNodes".semiAutoSplice.sequence.status.seqActive )
      wire#w1
      Coil( "Unit1.Em2.ControlNodes".semiAutoSplice."step".action1[2704] )
   END_RUNG
   RUNG wire#w1
      Coil( "Unit1.Em2.ControlNodes".semiAutoSplice."step".transition1[2704] )
   END_RUNG
   RUNG wire#w1
      Contact( "Unit1.Em2.ControlNodes".semiAutoSplice."step".transition1[2704] )
      { S7_Templates := "time_type := Time" } #statTonTimer[2704].TON(pt := #SeqDelayTime, et =>)
      Move(in := #JOB_27_STEP_05, out1 => "Unit1.Em2.ControlNodes".semiAutoSplice.sequence.status.nextStep)
   END_RUNG
   // the same network as SCL:
   "Unit1.Em2.ControlNodes".semiAutoSplice."step".action1[2704] := ("Unit1.Em2.ControlNodes".semiAutoSplice.sequence.status.currentStep = #JOB_27_STEP_04) AND "Unit1.Em2.ControlNodes".semiAutoSplice.sequence.status.seqActive;
   "Unit1.Em2.ControlNodes".semiAutoSplice."step".transition1[2704] := ("Unit1.Em2.ControlNodes".semiAutoSplice.sequence.status.currentStep = #JOB_27_STEP_04) AND "Unit1.Em2.ControlNodes".semiAutoSplice.sequence.status.seqActive;
   #statTonTimer[2704].TON(IN := ("Unit1.Em2.ControlNodes".semiAutoSplice.sequence.status.currentStep = #JOB_27_STEP_04) AND "Unit1.Em2.ControlNodes".semiAutoSplice.sequence.status.seqActive AND "Unit1.Em2.ControlNodes".semiAutoSplice."step".transition1[2704],
                           PT := #SeqDelayTime);
   IF #statTonTimer[2704].Q THEN
       "Unit1.Em2.ControlNodes".semiAutoSplice.sequence.status.nextStep := #JOB_27_STEP_05;
   END_IF;
END_REGION

REGION Network 137: Step[2705] :
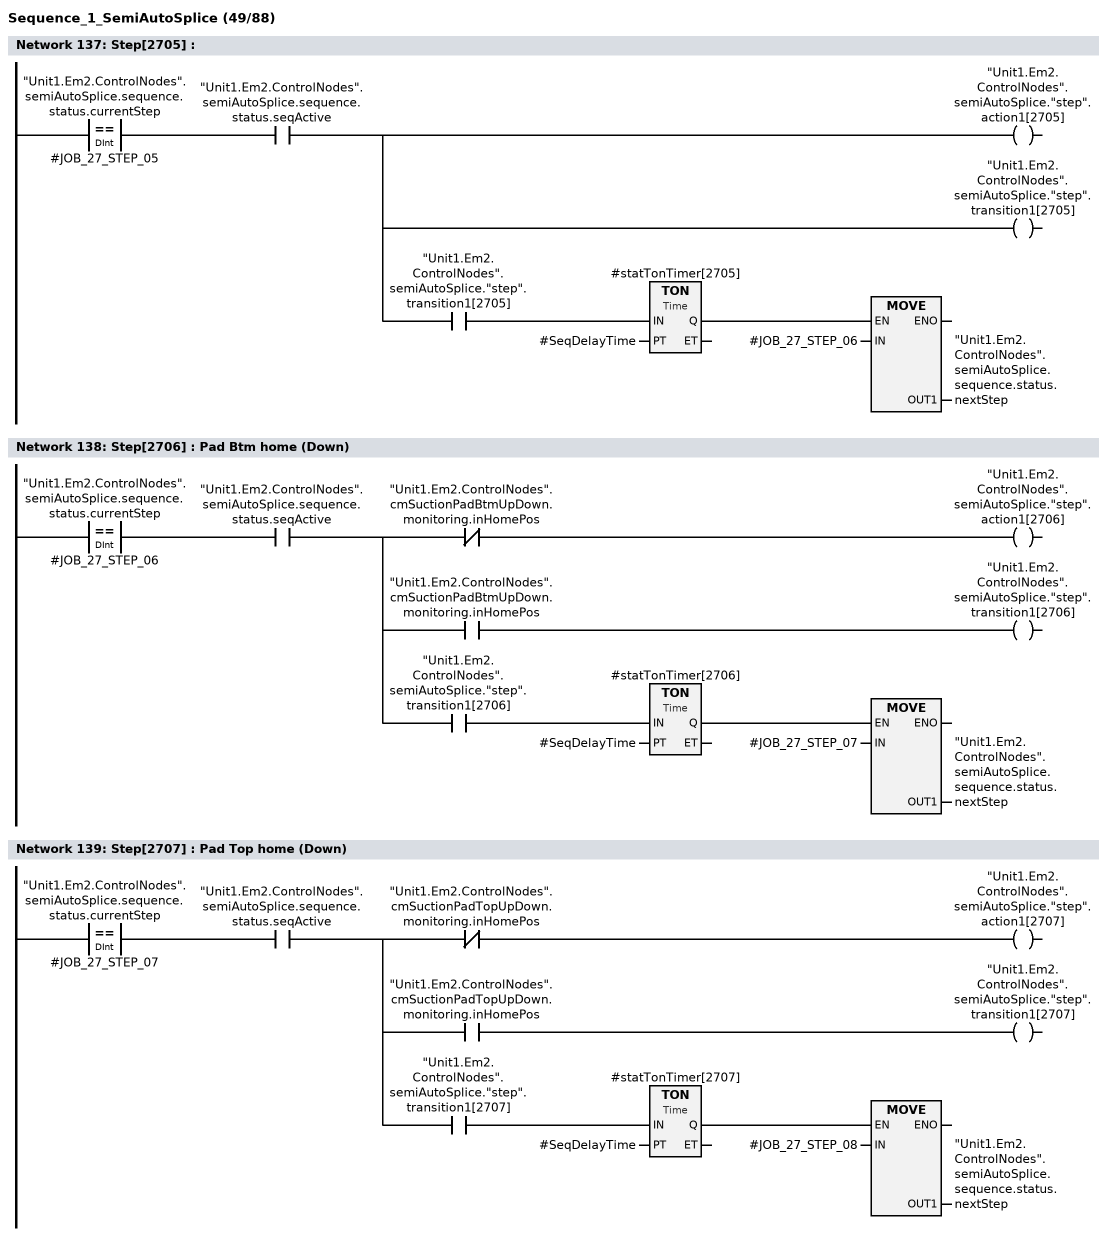
   RUNG wire#powerrail
      { S7_Templates := "SrcType := DInt" } EQ_Contact(in1 := "Unit1.Em2.ControlNodes".semiAutoSplice.sequence.status.currentStep, in2 := #JOB_27_STEP_05)
      Contact( "Unit1.Em2.ControlNodes".semiAutoSplice.sequence.status.seqActive )
      wire#w1
      Coil( "Unit1.Em2.ControlNodes".semiAutoSplice."step".action1[2705] )
   END_RUNG
   RUNG wire#w1
      Coil( "Unit1.Em2.ControlNodes".semiAutoSplice."step".transition1[2705] )
   END_RUNG
   RUNG wire#w1
      Contact( "Unit1.Em2.ControlNodes".semiAutoSplice."step".transition1[2705] )
      { S7_Templates := "time_type := Time" } #statTonTimer[2705].TON(pt := #SeqDelayTime, et =>)
      Move(in := #JOB_27_STEP_06, out1 => "Unit1.Em2.ControlNodes".semiAutoSplice.sequence.status.nextStep)
   END_RUNG
   // the same network as SCL:
   "Unit1.Em2.ControlNodes".semiAutoSplice."step".action1[2705] := ("Unit1.Em2.ControlNodes".semiAutoSplice.sequence.status.currentStep = #JOB_27_STEP_05) AND "Unit1.Em2.ControlNodes".semiAutoSplice.sequence.status.seqActive;
   "Unit1.Em2.ControlNodes".semiAutoSplice."step".transition1[2705] := ("Unit1.Em2.ControlNodes".semiAutoSplice.sequence.status.currentStep = #JOB_27_STEP_05) AND "Unit1.Em2.ControlNodes".semiAutoSplice.sequence.status.seqActive;
   #statTonTimer[2705].TON(IN := ("Unit1.Em2.ControlNodes".semiAutoSplice.sequence.status.currentStep = #JOB_27_STEP_05) AND "Unit1.Em2.ControlNodes".semiAutoSplice.sequence.status.seqActive AND "Unit1.Em2.ControlNodes".semiAutoSplice."step".transition1[2705],
                           PT := #SeqDelayTime);
   IF #statTonTimer[2705].Q THEN
       "Unit1.Em2.ControlNodes".semiAutoSplice.sequence.status.nextStep := #JOB_27_STEP_06;
   END_IF;
END_REGION

REGION Network 138: Step[2706] : Pad Btm home (Down)
   RUNG wire#powerrail
      { S7_Templates := "SrcType := DInt" } EQ_Contact(in1 := "Unit1.Em2.ControlNodes".semiAutoSplice.sequence.status.currentStep, in2 := #JOB_27_STEP_06)
      Contact( "Unit1.Em2.ControlNodes".semiAutoSplice.sequence.status.seqActive )
      wire#w1
      I_Contact( "Unit1.Em2.ControlNodes".cmSuctionPadBtmUpDown.monitoring.inHomePos )
      Coil( "Unit1.Em2.ControlNodes".semiAutoSplice."step".action1[2706] )
   END_RUNG
   RUNG wire#w1
      Contact( "Unit1.Em2.ControlNodes".cmSuctionPadBtmUpDown.monitoring.inHomePos )
      Coil( "Unit1.Em2.ControlNodes".semiAutoSplice."step".transition1[2706] )
   END_RUNG
   RUNG wire#w1
      Contact( "Unit1.Em2.ControlNodes".semiAutoSplice."step".transition1[2706] )
      { S7_Templates := "time_type := Time" } #statTonTimer[2706].TON(pt := #SeqDelayTime, et =>)
      Move(in := #JOB_27_STEP_07, out1 => "Unit1.Em2.ControlNodes".semiAutoSplice.sequence.status.nextStep)
   END_RUNG
   // the same network as SCL:
   #_w1 := ("Unit1.Em2.ControlNodes".semiAutoSplice.sequence.status.currentStep = #JOB_27_STEP_06) AND "Unit1.Em2.ControlNodes".semiAutoSplice.sequence.status.seqActive;
   "Unit1.Em2.ControlNodes".semiAutoSplice."step".action1[2706] := #_w1 AND NOT "Unit1.Em2.ControlNodes".cmSuctionPadBtmUpDown.monitoring.inHomePos;
   "Unit1.Em2.ControlNodes".semiAutoSplice."step".transition1[2706] := #_w1 AND "Unit1.Em2.ControlNodes".cmSuctionPadBtmUpDown.monitoring.inHomePos;
   #statTonTimer[2706].TON(IN := #_w1 AND "Unit1.Em2.ControlNodes".semiAutoSplice."step".transition1[2706],
                           PT := #SeqDelayTime);
   IF #statTonTimer[2706].Q THEN
       "Unit1.Em2.ControlNodes".semiAutoSplice.sequence.status.nextStep := #JOB_27_STEP_07;
   END_IF;
END_REGION

REGION Network 139: Step[2707] : Pad Top home (Down)
   RUNG wire#powerrail
      { S7_Templates := "SrcType := DInt" } EQ_Contact(in1 := "Unit1.Em2.ControlNodes".semiAutoSplice.sequence.status.currentStep, in2 := #JOB_27_STEP_07)
      Contact( "Unit1.Em2.ControlNodes".semiAutoSplice.sequence.status.seqActive )
      wire#w1
      I_Contact( "Unit1.Em2.ControlNodes".cmSuctionPadTopUpDown.monitoring.inHomePos )
      Coil( "Unit1.Em2.ControlNodes".semiAutoSplice."step".action1[2707] )
   END_RUNG
   RUNG wire#w1
      Contact( "Unit1.Em2.ControlNodes".cmSuctionPadTopUpDown.monitoring.inHomePos )
      Coil( "Unit1.Em2.ControlNodes".semiAutoSplice."step".transition1[2707] )
   END_RUNG
   RUNG wire#w1
      Contact( "Unit1.Em2.ControlNodes".semiAutoSplice."step".transition1[2707] )
      { S7_Templates := "time_type := Time" } #statTonTimer[2707].TON(pt := #SeqDelayTime, et =>)
      Move(in := #JOB_27_STEP_08, out1 => "Unit1.Em2.ControlNodes".semiAutoSplice.sequence.status.nextStep)
   END_RUNG
   // the same network as SCL:
   #_w1 := ("Unit1.Em2.ControlNodes".semiAutoSplice.sequence.status.currentStep = #JOB_27_STEP_07) AND "Unit1.Em2.ControlNodes".semiAutoSplice.sequence.status.seqActive;
   "Unit1.Em2.ControlNodes".semiAutoSplice."step".action1[2707] := #_w1 AND NOT "Unit1.Em2.ControlNodes".cmSuctionPadTopUpDown.monitoring.inHomePos;
   "Unit1.Em2.ControlNodes".semiAutoSplice."step".transition1[2707] := #_w1 AND "Unit1.Em2.ControlNodes".cmSuctionPadTopUpDown.monitoring.inHomePos;
   #statTonTimer[2707].TON(IN := #_w1 AND "Unit1.Em2.ControlNodes".semiAutoSplice."step".transition1[2707],
                           PT := #SeqDelayTime);
   IF #statTonTimer[2707].Q THEN
       "Unit1.Em2.ControlNodes".semiAutoSplice.sequence.status.nextStep := #JOB_27_STEP_08;
   END_IF;
END_REGION

REGION Network 140: Step[2708] : Complete
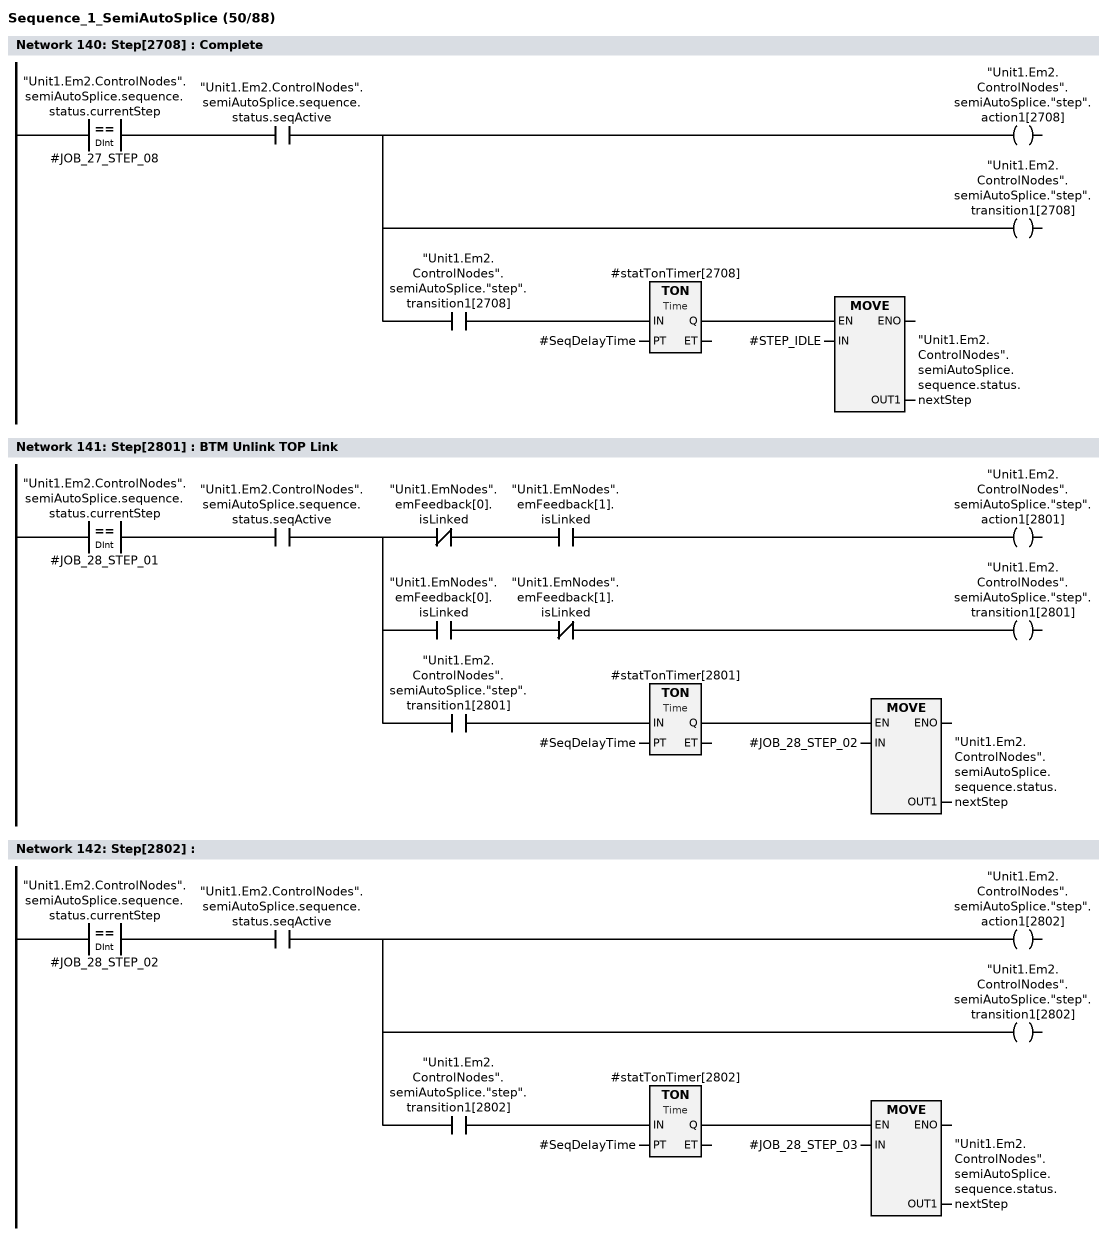
   RUNG wire#powerrail
      { S7_Templates := "SrcType := DInt" } EQ_Contact(in1 := "Unit1.Em2.ControlNodes".semiAutoSplice.sequence.status.currentStep, in2 := #JOB_27_STEP_08)
      Contact( "Unit1.Em2.ControlNodes".semiAutoSplice.sequence.status.seqActive )
      wire#w1
      Coil( "Unit1.Em2.ControlNodes".semiAutoSplice."step".action1[2708] )
   END_RUNG
   RUNG wire#w1
      Coil( "Unit1.Em2.ControlNodes".semiAutoSplice."step".transition1[2708] )
   END_RUNG
   RUNG wire#w1
      Contact( "Unit1.Em2.ControlNodes".semiAutoSplice."step".transition1[2708] )
      { S7_Templates := "time_type := Time" } #statTonTimer[2708].TON(pt := #SeqDelayTime, et =>)
      Move(in := #STEP_IDLE, out1 => "Unit1.Em2.ControlNodes".semiAutoSplice.sequence.status.nextStep)
   END_RUNG
   // the same network as SCL:
   "Unit1.Em2.ControlNodes".semiAutoSplice."step".action1[2708] := ("Unit1.Em2.ControlNodes".semiAutoSplice.sequence.status.currentStep = #JOB_27_STEP_08) AND "Unit1.Em2.ControlNodes".semiAutoSplice.sequence.status.seqActive;
   "Unit1.Em2.ControlNodes".semiAutoSplice."step".transition1[2708] := ("Unit1.Em2.ControlNodes".semiAutoSplice.sequence.status.currentStep = #JOB_27_STEP_08) AND "Unit1.Em2.ControlNodes".semiAutoSplice.sequence.status.seqActive;
   #statTonTimer[2708].TON(IN := ("Unit1.Em2.ControlNodes".semiAutoSplice.sequence.status.currentStep = #JOB_27_STEP_08) AND "Unit1.Em2.ControlNodes".semiAutoSplice.sequence.status.seqActive AND "Unit1.Em2.ControlNodes".semiAutoSplice."step".transition1[2708],
                           PT := #SeqDelayTime);
   IF #statTonTimer[2708].Q THEN
       "Unit1.Em2.ControlNodes".semiAutoSplice.sequence.status.nextStep := #STEP_IDLE;
   END_IF;
END_REGION

REGION Network 141: Step[2801] : BTM Unlink TOP Link
   RUNG wire#powerrail
      { S7_Templates := "SrcType := DInt" } EQ_Contact(in1 := "Unit1.Em2.ControlNodes".semiAutoSplice.sequence.status.currentStep, in2 := #JOB_28_STEP_01)
      Contact( "Unit1.Em2.ControlNodes".semiAutoSplice.sequence.status.seqActive )
      wire#w1
      I_Contact( "Unit1.EmNodes".emFeedback[0].isLinked )
      Contact( "Unit1.EmNodes".emFeedback[1].isLinked )
      Coil( "Unit1.Em2.ControlNodes".semiAutoSplice."step".action1[2801] )
   END_RUNG
   RUNG wire#w1
      Contact( "Unit1.EmNodes".emFeedback[0].isLinked )
      I_Contact( "Unit1.EmNodes".emFeedback[1].isLinked )
      Coil( "Unit1.Em2.ControlNodes".semiAutoSplice."step".transition1[2801] )
   END_RUNG
   RUNG wire#w1
      Contact( "Unit1.Em2.ControlNodes".semiAutoSplice."step".transition1[2801] )
      { S7_Templates := "time_type := Time" } #statTonTimer[2801].TON(pt := #SeqDelayTime, et =>)
      Move(in := #JOB_28_STEP_02, out1 => "Unit1.Em2.ControlNodes".semiAutoSplice.sequence.status.nextStep)
   END_RUNG
   // the same network as SCL:
   #_w1 := ("Unit1.Em2.ControlNodes".semiAutoSplice.sequence.status.currentStep = #JOB_28_STEP_01) AND "Unit1.Em2.ControlNodes".semiAutoSplice.sequence.status.seqActive;
   "Unit1.Em2.ControlNodes".semiAutoSplice."step".action1[2801] := #_w1 AND NOT "Unit1.EmNodes".emFeedback[0].isLinked AND "Unit1.EmNodes".emFeedback[1].isLinked;
   "Unit1.Em2.ControlNodes".semiAutoSplice."step".transition1[2801] := #_w1 AND "Unit1.EmNodes".emFeedback[0].isLinked AND NOT "Unit1.EmNodes".emFeedback[1].isLinked;
   #statTonTimer[2801].TON(IN := #_w1 AND "Unit1.Em2.ControlNodes".semiAutoSplice."step".transition1[2801],
                           PT := #SeqDelayTime);
   IF #statTonTimer[2801].Q THEN
       "Unit1.Em2.ControlNodes".semiAutoSplice.sequence.status.nextStep := #JOB_28_STEP_02;
   END_IF;
END_REGION

REGION Network 142: Step[2802] :
   RUNG wire#powerrail
      { S7_Templates := "SrcType := DInt" } EQ_Contact(in1 := "Unit1.Em2.ControlNodes".semiAutoSplice.sequence.status.currentStep, in2 := #JOB_28_STEP_02)
      Contact( "Unit1.Em2.ControlNodes".semiAutoSplice.sequence.status.seqActive )
      wire#w1
      Coil( "Unit1.Em2.ControlNodes".semiAutoSplice."step".action1[2802] )
   END_RUNG
   RUNG wire#w1
      Coil( "Unit1.Em2.ControlNodes".semiAutoSplice."step".transition1[2802] )
   END_RUNG
   RUNG wire#w1
      Contact( "Unit1.Em2.ControlNodes".semiAutoSplice."step".transition1[2802] )
      { S7_Templates := "time_type := Time" } #statTonTimer[2802].TON(pt := #SeqDelayTime, et =>)
      Move(in := #JOB_28_STEP_03, out1 => "Unit1.Em2.ControlNodes".semiAutoSplice.sequence.status.nextStep)
   END_RUNG
   // the same network as SCL:
   "Unit1.Em2.ControlNodes".semiAutoSplice."step".action1[2802] := ("Unit1.Em2.ControlNodes".semiAutoSplice.sequence.status.currentStep = #JOB_28_STEP_02) AND "Unit1.Em2.ControlNodes".semiAutoSplice.sequence.status.seqActive;
   "Unit1.Em2.ControlNodes".semiAutoSplice."step".transition1[2802] := ("Unit1.Em2.ControlNodes".semiAutoSplice.sequence.status.currentStep = #JOB_28_STEP_02) AND "Unit1.Em2.ControlNodes".semiAutoSplice.sequence.status.seqActive;
   #statTonTimer[2802].TON(IN := ("Unit1.Em2.ControlNodes".semiAutoSplice.sequence.status.currentStep = #JOB_28_STEP_02) AND "Unit1.Em2.ControlNodes".semiAutoSplice.sequence.status.seqActive AND "Unit1.Em2.ControlNodes".semiAutoSplice."step".transition1[2802],
                           PT := #SeqDelayTime);
   IF #statTonTimer[2802].Q THEN
       "Unit1.Em2.ControlNodes".semiAutoSplice.sequence.status.nextStep := #JOB_28_STEP_03;
   END_IF;
END_REGION

REGION Network 143: Step[2803] :
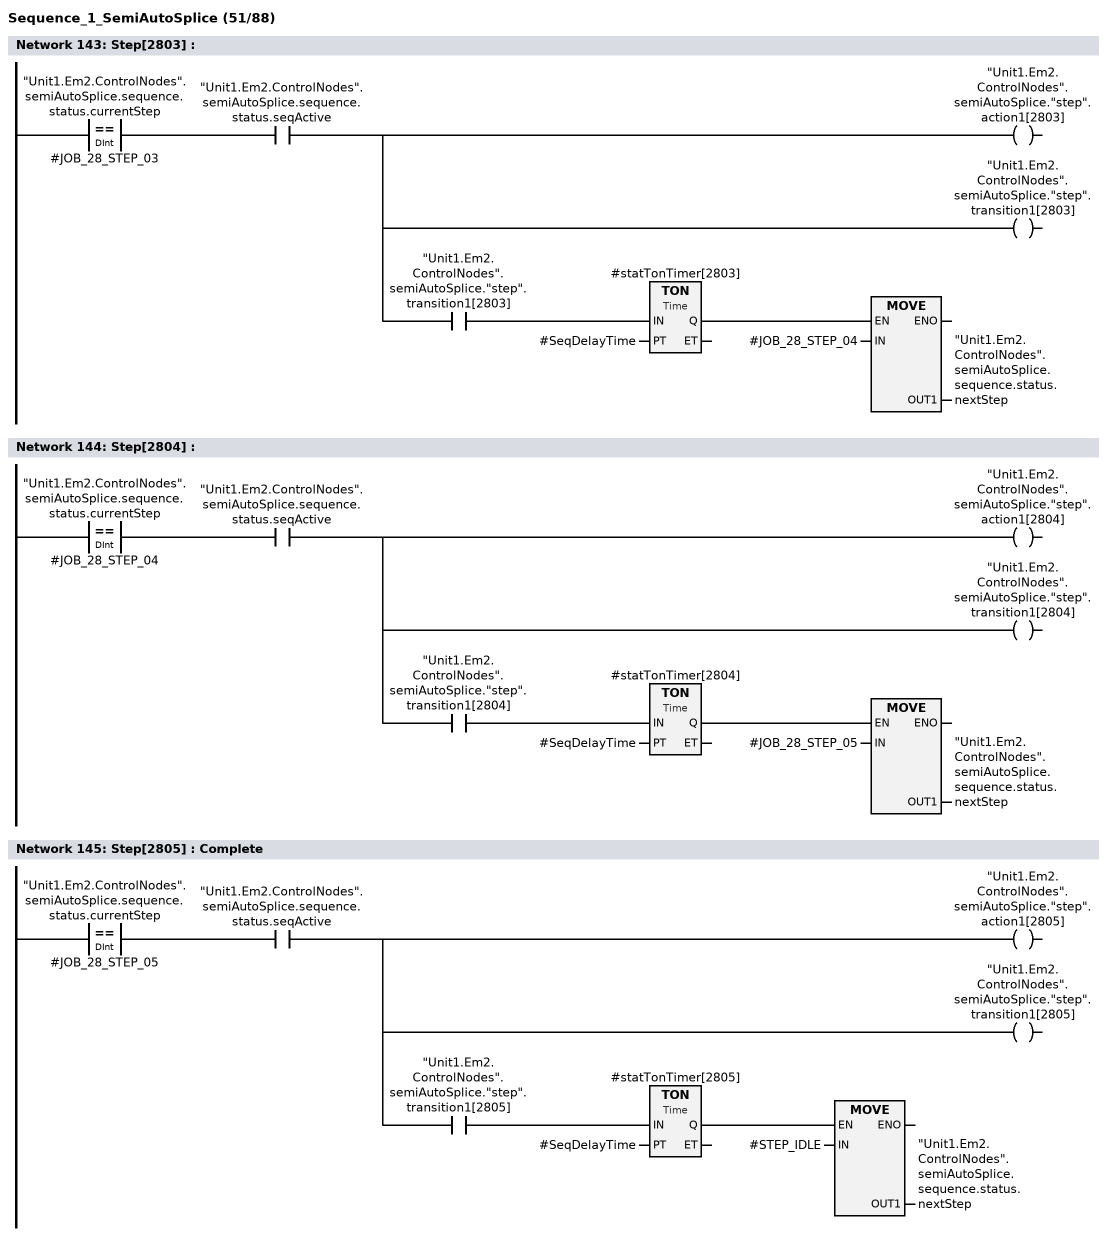
   RUNG wire#powerrail
      { S7_Templates := "SrcType := DInt" } EQ_Contact(in1 := "Unit1.Em2.ControlNodes".semiAutoSplice.sequence.status.currentStep, in2 := #JOB_28_STEP_03)
      Contact( "Unit1.Em2.ControlNodes".semiAutoSplice.sequence.status.seqActive )
      wire#w1
      Coil( "Unit1.Em2.ControlNodes".semiAutoSplice."step".action1[2803] )
   END_RUNG
   RUNG wire#w1
      Coil( "Unit1.Em2.ControlNodes".semiAutoSplice."step".transition1[2803] )
   END_RUNG
   RUNG wire#w1
      Contact( "Unit1.Em2.ControlNodes".semiAutoSplice."step".transition1[2803] )
      { S7_Templates := "time_type := Time" } #statTonTimer[2803].TON(pt := #SeqDelayTime, et =>)
      Move(in := #JOB_28_STEP_04, out1 => "Unit1.Em2.ControlNodes".semiAutoSplice.sequence.status.nextStep)
   END_RUNG
   // the same network as SCL:
   "Unit1.Em2.ControlNodes".semiAutoSplice."step".action1[2803] := ("Unit1.Em2.ControlNodes".semiAutoSplice.sequence.status.currentStep = #JOB_28_STEP_03) AND "Unit1.Em2.ControlNodes".semiAutoSplice.sequence.status.seqActive;
   "Unit1.Em2.ControlNodes".semiAutoSplice."step".transition1[2803] := ("Unit1.Em2.ControlNodes".semiAutoSplice.sequence.status.currentStep = #JOB_28_STEP_03) AND "Unit1.Em2.ControlNodes".semiAutoSplice.sequence.status.seqActive;
   #statTonTimer[2803].TON(IN := ("Unit1.Em2.ControlNodes".semiAutoSplice.sequence.status.currentStep = #JOB_28_STEP_03) AND "Unit1.Em2.ControlNodes".semiAutoSplice.sequence.status.seqActive AND "Unit1.Em2.ControlNodes".semiAutoSplice."step".transition1[2803],
                           PT := #SeqDelayTime);
   IF #statTonTimer[2803].Q THEN
       "Unit1.Em2.ControlNodes".semiAutoSplice.sequence.status.nextStep := #JOB_28_STEP_04;
   END_IF;
END_REGION

REGION Network 144: Step[2804] :
   RUNG wire#powerrail
      { S7_Templates := "SrcType := DInt" } EQ_Contact(in1 := "Unit1.Em2.ControlNodes".semiAutoSplice.sequence.status.currentStep, in2 := #JOB_28_STEP_04)
      Contact( "Unit1.Em2.ControlNodes".semiAutoSplice.sequence.status.seqActive )
      wire#w1
      Coil( "Unit1.Em2.ControlNodes".semiAutoSplice."step".action1[2804] )
   END_RUNG
   RUNG wire#w1
      Coil( "Unit1.Em2.ControlNodes".semiAutoSplice."step".transition1[2804] )
   END_RUNG
   RUNG wire#w1
      Contact( "Unit1.Em2.ControlNodes".semiAutoSplice."step".transition1[2804] )
      { S7_Templates := "time_type := Time" } #statTonTimer[2804].TON(pt := #SeqDelayTime, et =>)
      Move(in := #JOB_28_STEP_05, out1 => "Unit1.Em2.ControlNodes".semiAutoSplice.sequence.status.nextStep)
   END_RUNG
   // the same network as SCL:
   "Unit1.Em2.ControlNodes".semiAutoSplice."step".action1[2804] := ("Unit1.Em2.ControlNodes".semiAutoSplice.sequence.status.currentStep = #JOB_28_STEP_04) AND "Unit1.Em2.ControlNodes".semiAutoSplice.sequence.status.seqActive;
   "Unit1.Em2.ControlNodes".semiAutoSplice."step".transition1[2804] := ("Unit1.Em2.ControlNodes".semiAutoSplice.sequence.status.currentStep = #JOB_28_STEP_04) AND "Unit1.Em2.ControlNodes".semiAutoSplice.sequence.status.seqActive;
   #statTonTimer[2804].TON(IN := ("Unit1.Em2.ControlNodes".semiAutoSplice.sequence.status.currentStep = #JOB_28_STEP_04) AND "Unit1.Em2.ControlNodes".semiAutoSplice.sequence.status.seqActive AND "Unit1.Em2.ControlNodes".semiAutoSplice."step".transition1[2804],
                           PT := #SeqDelayTime);
   IF #statTonTimer[2804].Q THEN
       "Unit1.Em2.ControlNodes".semiAutoSplice.sequence.status.nextStep := #JOB_28_STEP_05;
   END_IF;
END_REGION

REGION Network 145: Step[2805] : Complete
   RUNG wire#powerrail
      { S7_Templates := "SrcType := DInt" } EQ_Contact(in1 := "Unit1.Em2.ControlNodes".semiAutoSplice.sequence.status.currentStep, in2 := #JOB_28_STEP_05)
      Contact( "Unit1.Em2.ControlNodes".semiAutoSplice.sequence.status.seqActive )
      wire#w1
      Coil( "Unit1.Em2.ControlNodes".semiAutoSplice."step".action1[2805] )
   END_RUNG
   RUNG wire#w1
      Coil( "Unit1.Em2.ControlNodes".semiAutoSplice."step".transition1[2805] )
   END_RUNG
   RUNG wire#w1
      Contact( "Unit1.Em2.ControlNodes".semiAutoSplice."step".transition1[2805] )
      { S7_Templates := "time_type := Time" } #statTonTimer[2805].TON(pt := #SeqDelayTime, et =>)
      Move(in := #STEP_IDLE, out1 => "Unit1.Em2.ControlNodes".semiAutoSplice.sequence.status.nextStep)
   END_RUNG
   // the same network as SCL:
   "Unit1.Em2.ControlNodes".semiAutoSplice."step".action1[2805] := ("Unit1.Em2.ControlNodes".semiAutoSplice.sequence.status.currentStep = #JOB_28_STEP_05) AND "Unit1.Em2.ControlNodes".semiAutoSplice.sequence.status.seqActive;
   "Unit1.Em2.ControlNodes".semiAutoSplice."step".transition1[2805] := ("Unit1.Em2.ControlNodes".semiAutoSplice.sequence.status.currentStep = #JOB_28_STEP_05) AND "Unit1.Em2.ControlNodes".semiAutoSplice.sequence.status.seqActive;
   #statTonTimer[2805].TON(IN := ("Unit1.Em2.ControlNodes".semiAutoSplice.sequence.status.currentStep = #JOB_28_STEP_05) AND "Unit1.Em2.ControlNodes".semiAutoSplice.sequence.status.seqActive AND "Unit1.Em2.ControlNodes".semiAutoSplice."step".transition1[2805],
                           PT := #SeqDelayTime);
   IF #statTonTimer[2805].Q THEN
       "Unit1.Em2.ControlNodes".semiAutoSplice.sequence.status.nextStep := #STEP_IDLE;
   END_IF;
END_REGION

